// CNC/4 MHT-Function/HLI3_FastMFunctionHandler
FUNCTION_BLOCK HLI3_FastMFunctionHandler
VAR_INPUT
	bForceOff			: BOOL;													(* Forces all bytes in the output array to be 00 and therefore to switch off the digital output *) 
	bReset				: BOOL;													(* Resets the digital output *)
	nFunctionNoOn		: UINT;													(* Specifies the M function number for switching the digital output on *) 
	nDelayOn			: DINT;													(* Specifies a delay time in [µs] for switching on the digital output *)
	nFunctionNoOff		: UINT;													(* Specifies the M function number for switching the digital output off *)
	nDelayOff			: DINT;													(* Specifies a delay time in [µs] for switching off the digital output *)
	stData				: ST_FastMFunctionData;									(* Structure provided by an instance of HLI3_FastMFunctionProvider *)
END_VAR
VAR_OUTPUT
	abyOutput			: ARRAY[0..MAX_FAST_M_FUNC_OUTPUT_IDX] OF BYTE;		(* Output array for a digital oversampling output terminal EL2262 *)  
END_VAR
VAR
	bSwitchOn			: BOOL;
	nSwitchOnOffset		: DINT;
	bSwitchOff			: BOOL;
	nSwitchOffOffset	: DINT;
	bStateChanged		: BOOL;
	bFirstCycle			: BOOL := TRUE;
	byStaticValue		: BYTE;
	byBitmask			: BYTE;
	nBits				: DINT;
	nBytes				: DINT;
	nLoop				: UINT;
	nQueuedCount		: UINT;
	
	eLastState			: E_FastMFunctionState := E_FastMFunctionState.OFF;
	stDequeued			: ST_FastMFunctionBufferItem;
	astQueue			: ARRAY[0..MAX_FAST_M_FUNC_QUEUE_IDX] OF ST_FastMFunctionBufferItem;
	
	fbRtrigReset		: Tc2_Standard.R_TRIG;
	CYCLE_TIME			: UINT := 1000;
END_VAR

(****************************************************************************************)
(* POU:		HLI3_FastMFunctionHandler                     								*)
(* Type:	FB																			*)
(* Author: 	RCH		                                             						*)
(* Date: 	14/10/29																	*)
(* Rev.: 	1.0                                               							*)
(* ------------------------------------------------------------------------------------ *)
(* Desc.:	Function block for handling the oversampled output on an EL2262. The 		*)
(*			output state will be derived from the occurance of two CNC M functions, 	*)
(*			which have to be configured with output method MOS_TS and which have to be	*)
(*			preprocessed by an instance of the HLI3_FastMFunctionProvider function 		*)
(*			block. The switch ON/OFF times can be delayed seperately.					*)					
(*																						*)
(*			THIS FB HAS TO BE CALLED CYCLICALLY IN A 1MS TASK AND THE EL2262 HAS TO 	*)
(*			FEATURE AN OVERSAMPLING FACTOR OF 1000 (125 BYTE) ==> 1µs == 1 bit!!!		*)
(* ------------------------------------------------------------------------------------ *)
(* Rev.:	1.1																			*)
(* Date:	15/05/05								                                   	*)
(* Author:	RCH																		 	*)
(* Desc.:	Fixed issues occured if more than 1 MOS_TS M function was programmed in a   *)
(*			single G-Code block.														*)
(* ------------------------------------------------------------------------------------ *)
(* Rev.:	<Enter revision number here>												*)
(* Date:	<Enter revision data here>				                                   	*)
(* Author:	<Enter author´s shortcut here>											 	*)
(* Desc.:	<Enter description here>													*)
(****************************************************************************************)

(****************************************************************************************)
(*	  						  Refresh buffered switch times 							*)
(****************************************************************************************)
THIS^.RefreshQueue(CYCLE_TIME);

(****************************************************************************************)
(*	  							 	  Reset output										*)
(****************************************************************************************)
fbRtrigReset(CLK:= bReset);

IF fbRtrigReset.Q THEN
	THIS^.ClearQueue();
	bStateChanged				:= TRUE;
	eLastState					:= E_FastMFunctionState.OFF;
END_IF

(****************************************************************************************)
(*	  					    Search for new switch on/off events 						*)
(****************************************************************************************)
bSwitchOn						:= FALSE;
nSwitchOnOffset					:= 0;
bSwitchOff						:= FALSE;
nSwitchOffOffset				:= 0;
nLoop							:= 0;

IF (stData.nFunctionCount > 0) AND (stData.bDataValid) THEN
	REPEAT
		IF (stData.astItem[nLoop].nFunctionNo = nFunctionNoOn) THEN
			bSwitchOn			:= TRUE;
			nSwitchOnOffset		:= stData.astItem[nLoop].nOffset;
		ELSIF (stData.astItem[nLoop].nFunctionNo = nFunctionNoOff) THEN
			bSwitchOff			:= TRUE;
			nSwitchOffOffset	:= stData.astItem[nLoop].nOffset;
		END_IF
	
		nLoop					:= nLoop + 1;
		
		UNTIL ((bSwitchOn AND bSwitchOff) OR (nLoop >= stData.nFunctionCount))
	END_REPEAT	
END_IF

(****************************************************************************************)
(*	  		Buffer found switch on/off events with correspondent switch times			*)
(****************************************************************************************)
IF bSwitchOn AND bSwitchOff THEN
	(* In case switch on and off events have been transmitted within the same cycle, 	*)
	(* order them according to their switch times!										*)
	IF ((nSwitchOnOffset + nDelayOn) < (nSwitchOffOffset + nDelayOff)) THEN
		THIS^.Enqueue(E_FastMFunctionState.ON, nSwitchOnOffset + nDelayOn);
		THIS^.Enqueue(E_FastMFunctionState.OFF, nSwitchOffOffset + nDelayOff); 
	ELSE
		THIS^.Enqueue(E_FastMFunctionState.OFF, nSwitchOffOffset + nDelayOff);
		THIS^.Enqueue(E_FastMFunctionState.ON, nSwitchOnOffset + nDelayOn);
	END_IF
ELSIF bSwitchOn THEN
	THIS^.Enqueue(E_FastMFunctionState.ON, nSwitchOnOffset + nDelayOn);
ELSIF bSwitchOff THEN
	THIS^.Enqueue(E_FastMFunctionState.OFF, nSwitchOffOffset + nDelayOff);
END_IF

(****************************************************************************************)
(*	  				  Set output array according to latest switch state					*)
(****************************************************************************************)
IF bStateChanged OR bFirstCycle THEN
	bStateChanged				:= FALSE;

	IF (eLastState = E_FastMFunctionState.OFF) THEN
		byStaticValue			:= 16#00;
	ELSIF (eLastState = E_FastMFunctionState.ON) THEN
		byStaticValue			:= 16#FF;
	END_IF
	
	Tc2_System.MEMSET(ADR(abyOutput[0]), byStaticValue, SIZEOF(abyOutput));
END_IF

(****************************************************************************************)
(*	  					  Dequeue switch events from the buffer							*)
(****************************************************************************************)
WHILE THIS^.DequeuingRequired DO
	stDequeued					:= THIS^.Dequeue();
	nBits 						:= stDequeued.nSwitchTime MOD 8;
	nBytes 						:= stDequeued.nSwitchTime / 8;
	bStateChanged				:= TRUE;
	IF (stDequeued.nSwitchTime < 0) OR (stDequeued.nSwitchTime > 1000) THEN
		;
	ELSE
		IF ((stDequeued.eState = E_FastMFunctionState.ON) AND (eLastState = E_FastMFunctionState.OFF)) THEN
			byBitmask			:= SHL(BYTE#255, nBits);
			abyOutput[nBytes]	:= abyOutput[nBytes] OR byBitmask;
			eLastState			:= E_FastMFunctionState.ON;
			Tc2_System.MEMSET(ADR(abyOutput[nBytes + 1]), 16#FF, MAX_FAST_M_FUNC_OUTPUT_IDX - nBytes);
		ELSIF ((stDequeued.eState = E_FastMFunctionState.OFF) AND (eLastState = E_FastMFunctionState.ON)) THEN
			byBitmask			:= SHR(BYTE#255, 8 - nBits);
			abyOutput[nBytes]	:= abyOutput[nBytes] AND byBitmask;
			eLastState			:= E_FastMFunctionState.OFF;
			Tc2_System.MEMSET(ADR(abyOutput[nBytes + 1]), 16#00, MAX_FAST_M_FUNC_OUTPUT_IDX - nBytes);
		END_IF
	END_IF
END_WHILE

(****************************************************************************************)
(*	  							   Reset first cycle indicator							*)
(****************************************************************************************)
bFirstCycle						:= FALSE;

METHOD ClearQueue
Tc2_System.MEMSET(ADR(astQueue), 16#00, SIZEOF(astQueue));
nQueuedCount := 0;
END_METHOD

METHOD Dequeue : ST_FastMFunctionBufferItem
VAR
	stReturn	: ST_FastMFunctionBufferItem;
END_VAR
IF (nQueuedCount > 0) THEN
	stReturn		:=	astQueue[0]; 
	Tc2_System.MEMMOVE(ADR(astQueue[0]), ADR(astQueue[1]), SIZEOF(astQueue) - SIZEOF(stReturn));
	
	nQueuedCount	:= nQueuedCount - 1;
	Dequeue			:= stReturn;
END_IF
END_METHOD

PROPERTY DequeuingRequired : BOOL
GET
DequeuingRequired	:= (nQueuedCount > 0) AND 
					   (astQueue[0].eState <> E_FastMFunctionState.EMPTY) AND
					   (astQueue[0].nSwitchTime < CYCLE_TIME);
END_GET
END_PROPERTY

METHOD Enqueue
VAR_INPUT
	eState			: E_FastMFunctionState;
	nSwitchTime		: DINT;
END_VAR
IF (nQueuedCount <= MAX_FAST_M_FUNC_OUTPUT_IDX) THEN
	astQueue[nQueuedCount].eState		:= eState;
	astQueue[nQueuedCount].nSwitchTime	:= nSwitchTime;
	nQueuedCount						:= nQueuedCount + 1;
END_IF
END_METHOD

METHOD RefreshQueue
VAR_INPUT
	nCycleTime: UINT;
END_VAR
IF (nQueuedCount > 0) THEN
	FOR nLoop := 0 TO (nQueuedCount - 1) DO
		astQueue[nLoop].nSwitchTime	:= astQueue[nLoop].nSwitchTime - nCycleTime;
	END_FOR
END_IF
END_METHOD

END_FUNCTION_BLOCK

// CNC/4 MHT-Function/HLI3_FastMFunctionProvider
FUNCTION_BLOCK HLI3_FastMFunctionProvider
VAR_INPUT
	nHliChanIdx				: UINT;													(* HLI channel index of the channel to check for new M functions *)
	anMFunctionNo			: ARRAY[0..MAX_FAST_M_FUNC_ITEM_IDX] OF UINT;			(* List of M functions munbers to handle *)
END_VAR
VAR_OUTPUT
	stData					: ST_FastMFunctionData;									(* Output structure containing informatione about the handled M functions and their execution offsets *)
	bUnknownChannelIndex	: BOOL;													(* TRUE if the given nHliChanIdx is unknown *)
END_VAR
VAR
	bExitAll				: BOOL;
	bFirstCycle				: BOOL := TRUE;
	byTaskIndex				: BYTE;
	nConfiguredFunctions	: UINT;
	nFunctionCount			: UINT;
	nLoop1					: UINT;
	nLoop2					: UINT;
	anMFunctionNoOld		: ARRAY[0..MAX_FAST_M_FUNC_ITEM_IDX] OF UINT;
	pChan					: POINTER TO HIGH_LEVEL_INTERFACE_CH;
	pData					: POINTER TO ST_FastMFunctionItem;
	pTechno					: POINTER TO Techno_Unit_Ch;
	pMHTechno				: POINTER TO HLI_M_H_Prozess;
	
	fbGetTaskIndex			: Tc2_System.GETCURTASKINDEX;
END_VAR

(****************************************************************************************)
(* POU:		HLI3_FastMFunctionProvider                     								*)
(* Type:	FB																			*)
(* Author: 	RCH		                                             						*)
(* Date: 	14/10/29																	*)
(* Rev.: 	1.0                                               							*)
(* ------------------------------------------------------------------------------------ *)
(* Desc.:	FB for handling CNC M functions contained in the input array				*)
(*			'anMFunctionNo'. These M functions have to be configured as MOS_TS. Their	*)
(*			metadata will be copied into the output structure 'stData' to be processed	*)
(*			by instances of the FB HLI3_FastMFunctionHandler!							*)				
(*																						*)
(*			THIS FB HAS TO BE CALLED CYCLICALLY IN A 1MS TASK!!!						*)
(* ------------------------------------------------------------------------------------ *)
(* Rev.:	1.1																			*)
(* Date:	15/05/05								                                   	*)
(* Author:	RCH																		 	*)
(* Desc.:	Fixed issues occured if more than 1 MOS_TS M function was programmed in a   *)
(*			single G-Code block.														*)
(* ------------------------------------------------------------------------------------ *)
(* Rev.:	<Enter revision number here>												*)
(* Date:	<Enter revision data here>				                                   	*)
(* Author:	<Enter author´s shortcut here>											 	*)
(* Desc.:	<Enter description here>													*)
(****************************************************************************************)

(****************************************************************************************)
(*	  Read current (PLC) task id and check whether the cycle time has been exceeded		*)
(****************************************************************************************)
IF bFirstCycle THEN
	fbGetTaskIndex
		(index				=> byTaskIndex);
END_IF

(****************************************************************************************)
(*								Initialize output structure								*)
(****************************************************************************************)
Tc2_System.MEMSET(ADR(stData), 16#00, SIZEOF(stData));

stData.bCycleTimeExceeded	:= TwinCAT_SystemInfoVarList._TaskInfo[byTaskIndex].CycleTimeExceeded;
stData.bDataValid			:= FALSE;
stData.nFunctionCount		:= 0;	

(****************************************************************************************)
(*	  					  Check existence of the given channel index					*)
(****************************************************************************************)
IF NOT HLI3_CheckChannelValid(nChannel := nHliChanIdx) THEN
	bUnknownChannelIndex	:=	TRUE; 
	RETURN;
ELSE
	bUnknownChannelIndex	:=	FALSE;
END_IF

(****************************************************************************************)
(*	  				  Determine the number of configured M functions					*)
(****************************************************************************************)
IF (Tc2_System.MEMCMP(ADR(anMFunctionNo), ADR(anMFunctionNoOld), SIZEOF(anMFunctionNo)) <> 0) THEN
	anMFunctionNoOld				:= anMFunctionNo;
	nConfiguredFunctions			:= 0;
	
	FOR nLoop1 := 0 TO MAX_FAST_M_FUNC_ITEM_IDX DO
		IF (anMFunctionNoOld[nLoop1] > 0) THEN
			nConfiguredFunctions	:= nConfiguredFunctions + 1;
		END_IF
	END_FOR
END_IF

(****************************************************************************************)
(*	  					  	Check occurances of M functions								*)
(****************************************************************************************)
stData.bDataValid					:= TRUE;
bFirstCycle							:= FALSE;

IF (gpCh[nHliChanIdx]^.used_units_std_sync_r = 0) THEN
	RETURN;
END_IF

pChan								:= gpCh[nHliChanIdx];
nFunctionCount						:= 0;
nLoop1 								:= 0;

FOR nLoop1 := 0 TO INT_TO_UINT(HLI_TU_CH_STD_SYNC_MAXIDX) DO
	IF pChan^.techno_unit_std_sync[nLoop1].please_rw AND (pChan^.techno_unit_std_sync[nLoop1].fkt_ctrl_r = Tc2_CncHli.HLI_INTF_M_FKT) THEN
		pTechno						:= ADR(pChan^.techno_unit_std_sync[nLoop1]);
		pMHTechno					:= ADR(pTechno^.attribut_r);	
		
		(* Check whether this FB has to handle the current M function *)
		FOR nLoop2 := 0 TO (nConfiguredFunctions - 1) DO
			IF (pMHTechno^.nr = anMFunctionNo[nLoop2]) THEN
				pData				:= ADR(stData.astItem[nFunctionCount]);
				pData^.nFunctionNo	:= anMFunctionNo[nLoop2];
				pData^.nOffset		:= pMHTechno^.zeit;
				pData^.nCycleCount	:= TwinCAT_SystemInfoVarList._TaskInfo[byTaskIndex].CycleCount;
				
				nFunctionCount		:= nFunctionCount + 1;
				
				pTechno^.please_rw	:= FALSE;
				pTechno^.done_w		:= TRUE;		
				EXIT;	
			END_IF					
		END_FOR
		
		IF (nFunctionCount >= nConfiguredFunctions) THEN
			EXIT;
		END_IF
	ELSIF NOT pChan^.techno_unit_std_sync[nLoop1].please_rw THEN
		EXIT;
	END_IF	
END_FOR

stData.nFunctionCount				:= nFunctionCount;

END_FUNCTION_BLOCK

// CNC/4 MHT-Function/HLI3_QuitAxisMFunction
FUNCTION HLI3_QuitAxisMFunction : BOOL
VAR_INPUT
	/// Number of axis 
	nHliAxisIdx: INT;
END_VAR
VAR
	/// Data of a M/H techno unit 
	pMHProcess: POINTER TO HLI_M_H_PROZESS;
	/// Data of a spindle unit 
	pSProcess: POINTER TO HLI_S_PROZESS;
	/// Data of a techno unit 
	pTProcess: POINTER TO HLI_T_PROZESS;
	/// local pointer to Data of actual Axis 
	pAxisData: POINTER TO HIGH_LEVEL_INTERFACE_AX;
	/// local pointer to actual techno unit 
	pActTechnoUnit: POINTER TO TECHNO_UNIT_AX;
	/// loop variable 
	idx: UINT;
	/// Index of axis specific technology function at HLI 
	nTechFctMaxIdx: UINT;
	/// basis id of a tool 
	nToolBasicId: UDINT;
	/// spindle movement command 
	SpdlMoveCmd: UINT;
	/// SpindleRevolution 
	Revolution: UDINT;
	/// SpindleRevolution 
	pRevolution: POINTER TO UDINT;
	/// Number of M-function 
	FuncNr: UDINT;
END_VAR

(* ========================================================= *)
(*    FUN: HLI_QuitAxisMFunction                             *)
(* --------------------------------------------------------- *)
(*   Desc:                                                   *)
(* Author: MK                                                *)
(*   Rev.: 1.1                                               *)
(*   Date: 18.07.2002                                        *)
(*       : 08.04.2005                                        *)
(* ========================================================= *)

HLI3_QuitAxisMFunction := FALSE;
IF NOT (HLI3_CheckAxisValid(nHliAxisIdx := nHliAxisIdx)) THEN
	RETURN;
END_IF


(* get pointer to Axis data *)
pAxisData := gpAx[nHliAxisIdx];

(* test if there are open synchronisations  *)
IF pAxisData^.used_units_std_sync_r > 0 THEN

	nTechFctMaxIdx := pAxisData^.used_units_std_sync_r - 1;

	FOR idx := 0 TO nTechFctMaxIdx DO
	
		(* get pointer to actual techno unit *)
		pActTechnoUnit := ADR(pAxisData^.techno_unit_std_sync[idx]);
	
		(* test if this M-function has to be acknowledged *)
		IF pActTechnoUnit^.please_rw = TRUE AND				(* request from CNC *)
			pActTechnoUnit^.done_w = FALSE					(* not acknowledged *)
		THEN
	
			IF pActTechnoUnit^.fkt_ctrl_r = HLI_INTF_M_FKT THEN
				(* Example: read number of M-function *)
				pMHProcess := ADR(pActTechnoUnit^.attribut_r.data[0]);
				FuncNr := pMHProcess^.nr;
				//ADSLOG(strMsg:='Axis acknowledge of M-function: %d', nDINT:=UDINT_TO_DINT(FuncNr), strArg:='');
			ELSE
				IF pActTechnoUnit^.fkt_ctrl_r = HLI_INTF_SPINDEL THEN (* spindle-fuction *)
					pSProcess := ADR(pActTechnoUnit^.attribut_r.data[0]);
	
					(* Example: read revolution of S-function *)
					Revolution := DINT_TO_UINT(pSProcess^.rev);
					//ADSLOG(strMsg:='Spindle S-function: %d', nDINT:=UDINT_TO_DINT(Revolution), strArg:='');
	
					(* Example: read number of S-function *)
					SpdlMoveCmd := pSProcess^.move_cmd;
					//ADSLOG(strMsg:='Spindle acknowledge of M-function: %d', nDINT:=SpdlMoveCmd, strArg:='');
				ELSE
					ADSLOGDINT( msgCtrlMask :=    ADSLOG_MSGTYPE_MSGBOX
					                           OR ADSLOG_MSGTYPE_LOG,
								msgFmtStr   := 'Axis acknowledge unknown type: %d',
								dintArg     := pActTechnoUnit^.fkt_ctrl_r);
				END_IF
			END_IF
	
			(* acknowledge this M-function *)
			pActTechnoUnit^.please_rw := FALSE;
			pActTechnoUnit^.done_w := TRUE;
	
			HLI3_QuitAxisMFunction := TRUE;
		END_IF
	END_FOR

END_IF

END_FUNCTION

// CNC/5 Variables/FB_ReadCNCVariables
FUNCTION_BLOCK FB_ReadCNCVariables
VAR_INPUT
	bEnable		:	BOOL ;	(* B *)
	nChanIdx	:   INT;
	eVariablesType : E_CNCVariablesType;
	tIntervall	:   TIME;
END_VAR

VAR_OUTPUT
	Done			:	BOOL;	(* B *)
	Busy			: 	BOOL;	(* E *)	
	Error			:	BOOL;	(* B *)
	ErrorID			:	UDINT;	(* E *) 
END_VAR

VAR_IN_OUT
	 stCNCVariablesViewer_Data : ARRAY[0..MAX_CNC_VAR_LIST_IDX] OF ST_CNCVariablesViewer_Data;
END_VAR

VAR	
	fbTrigger :	R_TRIG;
	fbReadNumber: ADSREAD;
	nParameterNumber : DINT;
		
	fbReadWrite: ADSRDWRT;	
	strVarName : STRING(96);	
	fVarValue  : LREAL;    
 	nIndex     : UDINT;
	nListIndex : UDINT;	
	
	nState	: INT;
	fbTimer : TON;

	nReadLength 	   : UDINT;
	
 	IDXOffsNumber	   : UDINT;
	IDXOffsNamebyIndex : UDINT;
	IDXOffsValuebyIndex : UDINT;	
	stCNCVariablesViewer_Data_Temp : ARRAY[0..MAX_CNC_VAR_LIST_IDX] OF ST_CNCVariablesViewer_Data;
		
	nVEType 				: DINT;
	nVESize 	 			: UDINT;
    nVEMaxIndex1 		   	: UDINT; 
    nVEMaxIndex2 		   	: UDINT;
	strVEVarName 			: STRING(255);	
	strVEDisplayVarName		: STRING(255);
	arrVEDescriptionInput  	: ARRAY[0..259] OF BYTE;
	arrVEOutput 			: ARRAY[0..2047] OF BYTE;
			
	nVEArrayIndex       	: UDINT;
	nListIndexArrayStart	: UDINT; 	
	
	strValue            : STRING(799);
			
	dummyBoolean		: BOOL;
	dummySInt			: SINT;
	dummyUSInt			: USINT;
	dummyInt            : INT;
	dummyUInt			: UINT;
	dummyDInt           : DINT;
	dummyUDInt          : UDINT;
	dummyLReal          : LREAL;
	dummyString         : STRING;
	dummyLargeString    : STRING(799);  

	eVariablesTypeOld : E_CNCVariablesType;
	
END_VAR

VAR CONSTANT
	IDXOffsPNumber  : UDINT := 16#2;	
	IDXOffsVLNumber : UDINT := 16#3;
	IDXOffsVPNumber : UDINT := 16#4;
	IDXOffsVSNumber : UDINT := 16#5;
			
	IDXOffsPNamebyIndex : UDINT := 16#1B;
	IDXOffsVLNamebyIndex : UDINT := 16#1E;
	IDXOffsVPNamebyIndex : UDINT := 16#21;
	IDXOffsVSNamebyIndex : UDINT := 16#24;		
	
	IDXOffsPValuebyIndex : UDINT := 16#1D;
	IDXOffsVLValuebyIndex : UDINT := 16#20;
	IDXOffsVPValuebyIndex : UDINT := 16#23;
	IDXOffsVSValuebyIndex : UDINT := 16#26;
	IDXOffsVEValuebyName : UDINT := 16#2E;		
END_VAR

(****************************************************************************************)
(* POU:		ReadCNCVariables                     										*)
(* Type:	FB																			*)
(* Author: 	TV , MiB                                       								*)
(* Date: 	20.01.2016, 19.12.2016														*)
(* Rev.: 	1.0                                              							*)
(* Rev.: 	1.1 MiB VStrings support (up to 800byte)           							*)
(* ------------------------------------------------------------------------------------ *)
(* Desc:	Description																	*)
(****************************************************************************************)

(****************************************************************************************)
(*	FB reads in P, V.P, V.L., V.S., V.E. Parameter from the CNC Kernel via ADS		    *)
(****************************************************************************************)

IF (NOT HLI3_CheckChannelValid(nChannel := nChanIdx)) THEN	
	RETURN; (* A b b r u c h *)
END_IF

IF 	NOT bEnable OR 
	eVariablesType = E_CNCVariablesType.none  OR
	(gpCh[0]^.channel_mc_control.mode_and_state.state_r.mode = HLI_IMCM_MANUAL_MODE AND eVariablesType <> E_CNCVariablesType.VE) OR
	(gpCh[nChanIdx]^.channel_mc_control.mode_and_state.state_r.state <> HLI_IMCM_PROCESS_ACTIVE AND 
	gpCh[nChanIdx]^.channel_mc_control.mode_and_state.state_r.state <>  HLI_IMCM_PROCESS_HOLD AND eVariablesType <> E_CNCVariablesType.VE) 
		
	THEN
		Tc2_System.MEMSET(ADR(stCNCVariablesViewer_Data),0,SIZEOF(stCNCVariablesViewer_Data));
		fbTrigger(CLK:= FALSE);
		nState := 0;  
	ELSE
		fbTrigger(CLK:= TRUE);	
END_IF

IF fbTrigger.Q OR eVariablesTypeOld <> eVariablesType THEN		
	fbReadNumber(READ:= FALSE);
	fbReadWrite(WRTRD:= FALSE);
	nIndex 		:= 1;	
	nListIndex  := 0;
	nState 		:= 1;
	Error		:= FALSE;	(* B *)
	ErrorID		:= 0;		(* E *) 
END_IF

IF nState <> 0 THEN
	Busy := TRUE;
END_IF

CASE nState OF
	
0:
;  
1: 
	Error		:= FALSE;	(* B *)
	ErrorID		:= 0;	(* E *)

	eVariablesTypeOld :=  eVariablesType;
 
	Tc2_System.MEMSET(ADR(stCNCVariablesViewer_Data_Temp),0,SIZEOF(stCNCVariablesViewer_Data_Temp));
	
   	IF (eVariablesType = E_CNCVariablesType.P) THEN
	      IDXOffsNumber 	 	:= IDXOffsPNumber;
		  IDXOffsNamebyIndex 	:= IDXOffsPNamebyIndex;
		  IDXOffsValuebyIndex 	:= IDXOffsPValuebyIndex;
		  nReadLength			:= 8;			  
	ELSIF (eVariablesType = E_CNCVariablesType.VL) THEN
		 IDXOffsNumber 		 	:=  IDXOffsVLNumber;
		 IDXOffsNamebyIndex  	:= IDXOffsVLNameByIndex;
		 IDXOffsValuebyIndex 	:= IDXOffsVLValuebyIndex;
		 nReadLength			:= 8;
	ELSIF (eVariablesType = E_CNCVariablesType.VP) THEN
		 IDXOffsNumber 		 	:=  IDXOffsVPNumber;
		 IDXOffsNamebyIndex  	:= IDXOffsVPNameByIndex;
		 IDXOffsValuebyIndex 	:= IDXOffsVPValuebyIndex;
		 nReadLength			:= 8;
	ELSIF (eVariablesType = E_CNCVariablesType.VS) THEN
		 IDXOffsNumber 		 	:=  IDXOffsVSNumber;
		 IDXOffsNamebyIndex  	:= IDXOffsVSNameByIndex;
		 IDXOffsValuebyIndex 	:= IDXOffsVSValuebyIndex;
		 nReadLength			:= 8;	
   	END_IF
				
	
	IF (eVariablesType <> E_CNCVariablesType.VE) THEN
		fbReadNumber(
			NETID:= , 
			PORT:= 552, 
			IDXGRP:= 16#22300 + INT_TO_UDINT(nChanIdx)+1, 
			IDXOFFS:= IDXOffsNumber, 
			LEN:= 4, 
			DESTADDR:= ADR(nParameterNumber), 
			READ:= TRUE, 
		);
		
		IF NOT fbReadNumber.Busy THEN
			IF fbReadNumber.Err	THEN
				Error := fbReadNumber.ERR;
				ErrorID := fbReadNumber.ERRID;
				nState := 99;
			ELSE			
				nState := nState + 1;				
			END_IF
		END_IF
	ELSE
		nState := 20;
	END_IF

2:	// Read Variablen Name	
	IF nParameterNumber > 0 THEN 
		fbReadWrite(
		NETID:= , 
		PORT:= 552, 
		IDXGRP:= 16#22300 + INT_TO_UDINT(nChanIdx)+1, 
		IDXOFFS:= IDXOffsNamebyIndex, 
		WRITELEN:= 4, 
		READLEN:= 96, 
		SRCADDR:= ADR(nIndex), 
		DESTADDR:=ADR(strVarName), 
		WRTRD:= TRUE);
	
		IF NOT fbReadWrite.Busy THEN
			IF fbReadWrite.Err	THEN
				Error := fbReadWrite.ERR;
				ErrorID := fbReadWrite.ERRID;
				nState := 99;
			ELSE					
				fbReadWrite(WRTRD:= FALSE);	
				nState := 3;							
			END_IF
		END_IF
	
	ELSE	
		nState := 99;
	END_IF
	
	
3:	// Read Variablen Value	P V.L. V.P. V.S	
		fbReadWrite(
		NETID:= , 
		PORT:= 552, 
		IDXGRP:= 16#22300 + INT_TO_UDINT(nChanIdx)+1, 
		IDXOFFS:= IDXOffsValuebyIndex, 
		WRITELEN:= 4, 
		READLEN:= nReadLength, 
		SRCADDR:= ADR(nIndex), 
		DESTADDR:=ADR(fVarValue), 
		WRTRD:= TRUE);
	
		IF NOT fbReadWrite.Busy THEN
			IF fbReadWrite.Err	THEN
				Error := fbReadWrite.ERR;
				ErrorID := fbReadWrite.ERRID;
				nState := 99;
			ELSE
				stCNCVariablesViewer_Data_Temp[nListIndex].strName := strVarName;
				stCNCVariablesViewer_Data_Temp[nListIndex].strValue := LREAL_TO_STRING(fVarValue);		
				nListIndex := nListIndex+1;								
				nState := 4;
			END_IF
		END_IF		
		
		
4:  
	IF nIndex < DINT_TO_UDINT(nParameterNumber) AND (nListIndex <= MAX_CNC_VAR_LIST_IDX) THEN
		fbReadWrite(WRTRD:= FALSE);
		//nListIndex := nListIndex+1; 
		nIndex := nIndex + 1;
		nState := 2;
	ELSE
			fbTimer(IN:=FALSE);
			nState := 60;
	END_IF

20:    	// Read V.E. Variable element number
		arrVEDescriptionInput[0] := 86; // V
		arrVEDescriptionInput[1] := 46; //.
		arrVEDescriptionInput[2] := 69; //E
		
		fbReadWrite(
			NETID:= , 
			PORT:= 552, 
			IDXGRP:= 16#22300 + INT_TO_UDINT(nChanIdx)+1, 
			IDXOFFS:= 16#44, 
			WRITELEN:= 256, 
			READLEN:= 4, 
			SRCADDR:= ADR(arrVEDescriptionInput), 
			DESTADDR:=ADR(nParameterNumber), 
			WRTRD:= TRUE);

			IF NOT fbReadWrite.Busy THEN
				IF fbReadWrite.Err	THEN
					Error := fbReadWrite.ERR;
					ErrorID := fbReadWrite.ERRID;
					nState := 99;
				ELSE
					fbReadWrite(WRTRD:= FALSE);
					IF nParameterNumber > 0 THEN	
						nIndex := 0;		
						nListIndexArrayStart := 0;
						nVEArrayIndex := 0;			
						nState := 21;					
					ELSE			
						fbTimer(IN:=FALSE);
						nState := 60;			
					END_IF
				END_IF	
			END_IF			
			
21:		// Read V.E. Variable description by index
		MEMCPY(ADR(arrVEDescriptionInput),ADR(nIndex),SIZEOF(nIndex));
		arrVEDescriptionInput[4] := 86; // V
		arrVEDescriptionInput[5] := 46; //.
		arrVEDescriptionInput[6] := 69; //E
		
		fbReadWrite(
			NETID:= , 
			PORT:= 552, 
			IDXGRP:= 16#22300 + INT_TO_UDINT(nChanIdx)+1, 
			IDXOFFS:= 16#45, 
			WRITELEN:= 260, 
			READLEN:= 2048, 
			SRCADDR:= ADR(arrVEDescriptionInput), 
			DESTADDR:=ADR(arrVEOutput), 
			WRTRD:= TRUE);
	
		IF NOT fbReadWrite.Busy THEN
			IF fbReadWrite.Err	THEN
				Error := fbReadWrite.ERR;
				ErrorID := fbReadWrite.ERRID;
				nState := 99;
			ELSE
				fbReadWrite(WRTRD:= FALSE);
				
				//MEMCPY(ADR(nHandle),ADR(arrByte3),SIZEOF(nHandle));
				MEMCPY(ADR(nVEType),ADR(arrVEOutput)+4,SIZEOF(nVEType));
				// MEMCPY(ADR(nAccess),ADR(arrByte3)+4+4,SIZEOF(nAccess));
				MEMCPY(ADR(nVESize),ADR(arrVEOutput)+4+4+4,SIZEOF(nVESize));
				MEMCPY(ADR(nVEMaxIndex1),ADR(arrVEOutput)+4+4+4+4,SIZEOF(nVEMaxIndex1));
				IF nVEMaxIndex1 <> 0 THEN
					MEMCPY(ADR(nVEMaxIndex2),ADR(arrVEOutput)+4+4+4+4+4,SIZEOF(nVEMaxIndex2));
					MEMCPY(ADR(strVEVarName),ADR(arrVEOutput)+4+4+4+4+4+4,SIZEOF(strVEVarName));
				ELSE
					MEMCPY(ADR(strVEVarName),ADR(arrVEOutput)+4+4+4+4+4,SIZEOF(strVEVarName));
				END_IF
												
				IF nVEMaxIndex1 > 0 THEN
					nListIndexArrayStart := nListIndex;
					FOR nVEArrayIndex := 0 TO nVEMaxIndex2-1 DO						
						strVEDisplayVarName := CONCAT(strVEVarName,'[');
						strVEDisplayVarName := CONCAT(strVEDisplayVarName,UDINT_TO_STRING(nVEArrayIndex));
						strVEDisplayVarName := CONCAT(strVEDisplayVarName,']');			
						stCNCVariablesViewer_Data_Temp[nListIndex].strName := strVEDisplayVarName;
						IF (nListIndex < MAX_CNC_VAR_LIST_IDX) THEN
							nListIndex := nListIndex+1;
						ELSE
							EXIT;
						END_IF
							
					END_FOR	
					   nVEArrayIndex := 0;
					   nListIndex := nListIndexArrayStart;
					   nState := 25;											
				ELSE			
					nVEArrayIndex := 0;
					stCNCVariablesViewer_Data_Temp[nListIndex].strName := strVEVarName;						
					nState := 25;
				END_IF						
			END_IF
		END_IF	
		
25:		// Read Value By Name	
		IF nVEMaxIndex1 = 0 THEN			
			strVEVarName := stCNCVariablesViewer_Data_Temp[nListIndex].strName;
		ELSE
			strVEVarName := stCNCVariablesViewer_Data_Temp[nListIndex+nVEArrayIndex].strName ;
		END_IF		
							
		fbReadWrite(
		NETID:= , 
		PORT:= 552, 
		IDXGRP:= 16#22300 + INT_TO_UDINT(nChanIdx)+1, 
		IDXOFFS:= 16#48, 
		WRITELEN:= SIZEOF(strVEVarName), 
		READLEN:= 2048, 
		SRCADDR:= ADR(strVEVarName), 
		DESTADDR:=ADR(arrVEOutput), 
		WRTRD:= TRUE);
		
		IF NOT fbReadWrite.Busy THEN
			IF fbReadWrite.Err	THEN
				Error := fbReadWrite.ERR;
				ErrorID := fbReadWrite.ERRID;
				nState := 99;
			ELSE	
						
				IF nVEType = E_VEVariablesType.BOOLEAN THEN 
					MEMCPY(ADR(dummyBoolean),ADR(arrVEOutput),1);
					strValue := BOOL_TO_STRING(dummyBoolean);
				ELSIF nVEType = E_VEVariablesType.UNS08 THEN
					MEMCPY(ADR(dummyUSInt),ADR(arrVEOutput),1);
					strValue := USINT_TO_STRING(dummyUSInt);
				ELSIF nVEType = E_VEVariablesType.SGN08 THEN
					MEMCPY(ADR(dummySInt),ADR(arrVEOutput),1);
					strValue := SINT_TO_STRING(dummySInt);
				ELSIF nVEType = E_VEVariablesType.UNS16 THEN
					MEMCPY(ADR(dummyUInt),ADR(arrVEOutput),2);
					strValue := UINT_TO_STRING(dummyUInt);
				ELSIF nVEType = E_VEVariablesType.SGN16 THEN
					MEMCPY(ADR(dummyInt),ADR(arrVEOutput),2);
					strValue := INT_TO_STRING(dummyInt);
				ELSIF nVEType = E_VEVariablesType.UNS32 THEN
					MEMCPY(ADR(dummyUDInt),ADR(arrVEOutput),4);
					strValue := UDINT_TO_STRING(dummyUDInt);
				ELSIF nVEType = E_VEVariablesType.SGN32 THEN
					MEMCPY(ADR(dummyDInt),ADR(arrVEOutput),4);
					strValue := DINT_TO_STRING(dummyDInt);
				ELSIF nVEType = E_VEVariablesType.REAL64 THEN
					MEMCPY(ADR(dummyLReal),ADR(arrVEOutput),8);
					strValue := LREAL_TO_STRING(dummyLReal);						
				ELSIF nVEType = E_VEVariablesType.VESTRING THEN					 									
					MEMCPY(ADR(dummyLargeString),ADR(arrVEOutput),nVESize-1);
					strValue := dummyLargeString;
				ELSE
					nState := 99;
				END_IF				
				
				nState := 26;	
			END_IF
		END_IF	
		
26:
		stCNCVariablesViewer_Data_Temp[nListIndex+nVEArrayIndex].strValue := strValue;									
										
		IF nVEArrayIndex < nVEMaxIndex2-1 AND  nVEMaxIndex1 <> 0 THEN
			fbReadWrite(WRTRD:= FALSE);
			nVEArrayIndex := nVEArrayIndex +1;
			IF (nListIndex+nVEArrayIndex <= MAX_CNC_VAR_LIST_IDX) THEN
				nState := 25;
			ELSE
				nState := 60;
			END_IF
		ELSE
			IF (nListIndex <= MAX_CNC_VAR_LIST_IDX) THEN
				nListIndex := nListIndex+nVEArrayIndex +1;
				nState := 30;
			ELSE
				nState := 60;
			END_IF		
			
		END_IF
		
30:  
	IF nIndex < DINT_TO_UDINT(nParameterNumber-1) THEN
		fbReadWrite(WRTRD:= FALSE);		 
		nIndex := nIndex + 1;
		nState := 21;
	ELSE
		fbReadWrite(WRTRD:= FALSE);				
		fbTimer(IN:=FALSE);			
		nState := 60;
	END_IF

60:
	// Output
	Tc2_System.MEMCPY(ADR(stCNCVariablesViewer_Data),ADR(stCNCVariablesViewer_Data_Temp),SIZEOF(stCNCVariablesViewer_Data_Temp));
	fbTimer(IN:=TRUE , PT:=tIntervall);	
	IF fbTimer.Q THEN
		fbReadNumber(READ:= FALSE);
		fbReadWrite(WRTRD:= FALSE);
		nListIndex := 0;
		nIndex := 1;
		nState := 1;
	END_IF

99: // Error 
	nIndex := 1;
	nListIndex := 0;
	fbReadNumber(READ:= FALSE);
	fbReadWrite(WRTRD:= FALSE);
	fbTimer(IN:=FALSE);
	nState := 60;			
END_CASE

END_FUNCTION_BLOCK

// CNC/5 Variables/HLI3_GetVEChannelBooleanValue
FUNCTION HLI3_GetVEChannelBooleanValue : BOOL
VAR_INPUT
	/// HLI Channel Index
	nChanIdx: INT;
	/// Index of variable  range 1 ...     HLI_VE_VALUEMAX 
	nVEIndex: DINT;
	/// Array index. 0 if no array 
	nArrayIndex: DINT := 0;
	/// serves acess to the global variable array 
	bGlobal: BOOL;
END_VAR
VAR
	pVeData: POINTER TO VEData := 0;
	/// Size of the datatype of the returned value 
	iDatatypeSize: DINT;
	ptr: POINTER TO BOOL;
	ChIdx: UDINT;
	SizeField: DINT := 0;
END_VAR

(* ========================================================= *)
(*    FUN: GetVEChannelDINTValue                            *)
(* --------------------------------------------------------- *)
(*   Desc: Reads a V.E.Variable of Boolean                   *)
(* 	 Author: CL  / TV                                        *)
(*   Date: 16.05.2006                                        *)
(*   Last: 05.12.2013                                        *)
(*   Rev.: 1.3                                               *)
(* ========================================================= *)

IF  nVEIndex >= 0 AND
	nArrayIndex >= 0 THEN

	(* test if channel specific or global *)
	IF bGlobal = FALSE  THEN
		IF NOT HLI3_CheckChannelValid(nChannel := nChanIdx) THEN
			RETURN;
		END_IF
				
		pVeData := gpVECh[nChanIdx];
	ELSE
		pVeData := gpVEGlobal;
	END_IF

	IF pVeData <> 0 THEN
		IF pVeData <> 0 THEN
			iDatatypeSize := SIZEOF(ptr^);
                         	ptr := pVeData +  24  * nVEIndex + (iDatatypeSize * nArrayIndex);
                           HLI3_GetVEChannelBooleanValue := ptr^; (* successfully completed return *)
                END_IF
	END_IF
END_IF

END_FUNCTION

// CNC/5 Variables/HLI3_GetVEChannelDIntValue
FUNCTION HLI3_GetVEChannelDIntValue : DINT
VAR_INPUT
	/// HLI Channel Index 
	nChanIdx: INT;
	/// Index of variable  range 1 ...     HLI_VE_VALUEMAX 
	nVEIndex: DINT;
	/// Array index. 0 if no array 
	nArrayIndex: DINT := 0;
	/// serves acess to the global variable array 
	bGlobal: BOOL;
END_VAR
VAR
	pVeData: POINTER TO VEData := 0;
	/// Size of the datatype of the returned value 
	iDatatypeSize: DINT;
	ptr: POINTER TO DINT;
	ChIdx: UDINT;
	SizeField: DINT := 0;
END_VAR

(* ========================================================= *)
(*    FUN: GetVEChannelDINTValue                            *)
(* --------------------------------------------------------- *)
(*   Desc: Reads a V.E.Variable of DINT                    *)
(* 	 Author: CL  / TV                                        *)
(*   Date: 16.05.2006                                        *)
(*   Last: 28.01.2013                                        *)
(*   Rev.: 1.3                                               *)
(* ========================================================= *)

IF  nVEIndex >= 0 AND
	nArrayIndex >= 0 THEN

	(* test if channel specific or global *)
	IF bGlobal = FALSE  THEN
		IF NOT HLI3_CheckChannelValid(nChannel := nChanIdx) THEN
			RETURN;
		END_IF
				
		pVeData := gpVECh[nChanIdx];
	ELSE
		pVeData := gpVEGlobal;
	END_IF

	IF pVeData <> 0 THEN
		IF pVeData <> 0 THEN
			iDatatypeSize := SIZEOF(ptr^);
                         	ptr := pVeData +  24  * nVEIndex + (iDatatypeSize * nArrayIndex);
                           HLI3_GetVEChannelDIntValue := ptr^; (* successfully completed return *)
                END_IF
	END_IF
END_IF

END_FUNCTION

// CNC/5 Variables/HLI3_GetVEChannelLRealValue
FUNCTION HLI3_GetVEChannelLRealValue : LREAL
VAR_INPUT
	/// HLI Channel Index
	nChanIdx: INT;
	/// Index of variable  range 1 ...     HLI_VE_VALUEMAX 
	nVEIndex: DINT;
	/// Array index. 0 if no array 
	nArrayIndex: DINT := 0;
	/// serves acess to the global variable array 
	bGlobal: BOOL;
END_VAR
VAR
	pVeData: POINTER TO VEData := 0;
	/// Size of the datatype of the returned value 
	iDatatypeSize: DINT;
	ptr: POINTER TO LREAL;
	ChIdx: UDINT;
	SizeField: DINT := 0;
END_VAR

(* ========================================================= *)
(*    FUN: GetVEChannelLrealValue                            *)
(* --------------------------------------------------------- *)
(*   Desc: Reads a V.E.Variable of REAL64                    *)
(* 	 Author: CL  / TV                                        *)
(*   Date: 16.05.2006                                        *)
(*   Last: 28.01.2013                                        *)
(*   Rev.: 1.3                                               *)
(* ========================================================= *)

IF  nVEIndex >= 0 AND
	nArrayIndex >= 0 THEN

	(* test if channel specific or global *)
	IF bGlobal = FALSE  THEN
		IF NOT HLI3_CheckChannelValid(nChannel := nChanIdx) THEN
			RETURN;
		END_IF
				
		pVeData := gpVECh[nChanIdx];
	ELSE
		pVeData := gpVEGlobal;
	END_IF

	IF pVeData <> 0 THEN
		IF pVeData <> 0 THEN
			iDatatypeSize := SIZEOF(ptr^);
                         	ptr := pVeData +  24  * nVEIndex + (iDatatypeSize * nArrayIndex);
                           HLI3_GetVEChannelLRealValue := ptr^; (* successfully completed return *)
                END_IF
	END_IF
END_IF

END_FUNCTION

// CNC/5 Variables/HLI3_GetVEChannelStringValue
FUNCTION HLI3_GetVEChannelStringValue : STRING(23)
VAR_INPUT
	/// HLI Channel Index
	nChanIdx: INT;
	/// Index of variable  range 1 ...     HLI_VE_VALUEMAX 
	nVEIndex: DINT;
	/// Array index. 0 if no array 
	nArrayIndex: DINT := 0;
	/// serves acess to the global variable array 
	bGlobal: BOOL;
END_VAR
VAR
	pVeData: POINTER TO VEData := 0;
	/// Size of the datatype of the returned value 
	iDatatypeSize: DINT;
	ptr: POINTER TO STRING(24);
	ChIdx: INT;
END_VAR

(* ========================================================= *)
(*    FUN: GetVEChannelStringValue                           *)
(* --------------------------------------------------------- *)
(*   Desc: Reads a V.E.Variable of STRING                    *)
(* 	 Author: CL / TV                                         *)
(*   Date: 16.05.2006                                        *)
(*   Last: 28.01.013                                        *)
(*   Rev.: 1.1                                               *)
(* ========================================================= *)

(* Config Example
	VAR[0].name                                           StringValue
	VAR[0].index                                           1
	VAR[0].TYPE                                           STRING
	VAR[0].scope                                          GLOBAL
	VAR[0].synchronisation                                TRUE
	VAR[0].access_rights                                  READ_WRITE
	VAR[0].array_size                                     21
	VAR[0].size                                           24
	VAR[0].create_hmi_interface                           0
*)

IF  nVEIndex >= 0 AND
	nArrayIndex >= 0 THEN

	(* test if channel specific or global *)
	IF bGlobal = FALSE  THEN
		IF NOT HLI3_CheckChannelValid(nChannel := nChanIdx) THEN
			RETURN;
		END_IF
		pVeData := gpVECh[nChanIdx];
	ELSE
		pVeData := gpVEGlobal;
	END_IF

	IF pVeData <> 0 THEN
		 IF pVeData <> 0 THEN
			iDatatypeSize := SIZEOF(ptr^);
			iDatatypeSize := 24;
            ptr := pVeData +  24  * nVEIndex + (iDatatypeSize * nArrayIndex);
            HLI3_GetVEChannelStringValue := ptr^; (* successfully completed return *)
         END_IF
	END_IF
END_IF

END_FUNCTION

// CNC/5 Variables/HLI3_LinkVEChannelStructure
FUNCTION HLI3_LinkVEChannelStructure : POINTER TO DWORD
VAR_INPUT
	/// HLI Channel Index 
	nChanIdx: INT;	
	/// serves acess to the global variable array 
	bGlobal: BOOL;
END_VAR
VAR
	pVeData: POINTER TO VEData := 0;
	ptr: POINTER TO DWORD;
	ChIdx: UDINT;
	nVEIndex: POINTER TO DWORD;
END_VAR

(* ========================================================= *)
(*    FUN: LinkVEChannelStructure                            *)
(* --------------------------------------------------------- *)
(*   Desc: Link VE variable to the memory of the CNC         *)
(*   Author: CL, MK                                            *)
(*   Date: 16.05.2006                                        *)
(*   Rev.: 1.3                                               *)
(*       : MK  access changed                                *)
(*		   1.2												 *)
(*		   MiB 7.11.2012 check zero pointers				 *)
(*		   TV 19.08.2015 Input Parm. nIndex removed          *) 
(* ========================================================= *)

	(* test if channel specific or global *)
     IF bGlobal THEN
    	IF gpVEGlobal = 0  THEN   (* check for  zero pointer *)
        	RETURN; (* Cancel *)
        END_IF
			pVeData := gpVEGlobal;
	 ELSE
		IF NOT HLI3_CheckChannelValid(nChannel := nChanIdx) THEN
			RETURN;
		END_IF
							
		pVeData := gpVECh[nChanIdx];
	END_IF 

	IF pVeData <> 0 THEN
    	ptr := pVeData;
		HLI3_LinkVEChannelStructure := ptr; (* successfully completed return *)
	END_IF

END_FUNCTION

// CNC/5 Variables/HLI3_SetVEChannelBooleanValue
FUNCTION HLI3_SetVEChannelBooleanValue : BOOL
VAR_INPUT
	/// HLI Channel Index
	nChanIdx: INT;
	/// Index of variable  range 1 ...     HLI_VE_VALUEMAX 
	nVEIndex: DINT;
	/// Array index. 0 if no array 
	nArrayIndex: DINT := 0;
	/// serves acess to the global variable array 
	bGlobal: BOOL;
	/// Value to be written 
	val: BOOL;
END_VAR
VAR
	pVeData: POINTER TO VEData := 0;
	/// Size of the datatype of the returned value 
	iDatatypeSize: DINT;
	ptr: POINTER TO BOOL;
	ChIdx: UDINT;
	SizeField: DINT := 0;
END_VAR

(* ========================================================= *)
(*    FUN: SetVEChannelDIntValue                           *)
(* --------------------------------------------------------- *)
(*   Desc: Writes a V.E.Variable of REAL64                    *)
(* 	 Author: CL  / TV                                        *)
(*   Date: 16.05.2006                                        *)
(*   Last: 05.12.2013                                        *)
(*   Rev.: 1.3                                               *)
(* ========================================================= *)

IF  nVEIndex >= 0 AND
	nArrayIndex >= 0 THEN

	(* test if channel specific or global *)
	IF bGlobal = FALSE  THEN
		IF NOT HLI3_CheckChannelValid(nChannel := nChanIdx) THEN
			RETURN;
		END_IF
				
		pVeData := gpVECh[nChanIdx];
	ELSE
		pVeData := gpVEGlobal;
	END_IF

	IF pVeData <> 0 THEN
		IF pVeData <> 0 THEN
			iDatatypeSize := SIZEOF(ptr^);
            ptr := pVeData +  24  * nVEIndex + (iDatatypeSize * nArrayIndex);
			ptr^:=val;
            HLI3_SetVEChannelBOOLeanValue := TRUE; (* successfully completed return *)						  						   
       	END_IF
	END_IF
END_IF

END_FUNCTION

// CNC/5 Variables/HLI3_SetVEChannelDIntValue
FUNCTION HLI3_SetVEChannelDIntValue : BOOL
VAR_INPUT
	/// HLI Channel Index
	nChanIdx: INT;
	/// Index of variable  range 1 ...     HLI_VE_VALUEMAX 
	nVEIndex: DINT;
	/// Array index. 0 if no array 
	nArrayIndex: DINT := 0;
	/// serves acess to the global variable array 
	bGlobal: BOOL;
	/// Value to be written 
	val: DINT;
END_VAR
VAR
	pVeData: POINTER TO VEData := 0;
	/// Size of the datatype of the returned value 
	iDatatypeSize: DINT;
	ptr: POINTER TO DINT;
	ChIdx: UDINT;
	SizeField: DINT := 0;
END_VAR

(* ========================================================= *)
(*    FUN: SetVEChannelDIntValue                           *)
(* --------------------------------------------------------- *)
(*   Desc: Writes a V.E.Variable of REAL64                    *)
(* 	 Author: CL  / TV                                        *)
(*   Date: 16.05.2006                                        *)
(*   Last: 28.01.2013                                        *)
(*   Rev.: 1.3                                               *)
(* ========================================================= *)

IF  nVEIndex >= 0 AND
	nArrayIndex >= 0 THEN

	(* test if channel specific or global *)
	IF bGlobal = FALSE  THEN
		IF NOT HLI3_CheckChannelValid(nChannel := nChanIdx) THEN
			RETURN;
		END_IF
				
		pVeData := gpVECh[nChanIdx];
	ELSE
		pVeData := gpVEGlobal;
	END_IF

	IF pVeData <> 0 THEN
		IF pVeData <> 0 THEN
			iDatatypeSize := SIZEOF(ptr^);
            ptr := pVeData +  24  * nVEIndex + (iDatatypeSize * nArrayIndex);
			ptr^:=val;
            HLI3_SetVEChannelDIntValue := TRUE; (* successfully completed return *)						  						   
       	END_IF
	END_IF
END_IF

END_FUNCTION

// CNC/5 Variables/HLI3_SetVEChannelLRealValue
FUNCTION HLI3_SetVEChannelLRealValue : BOOL
VAR_INPUT
	/// HLI Channel Index
	nChanIdx: INT;
	/// Index of variable  range 1 ...     HLI_VE_VALUEMAX 
	nVEIndex: DINT;
	/// Array index. 0 if no array 
	nArrayIndex: DINT := 0;
	/// serves acess to the global variable array 
	bGlobal: BOOL;
	/// Value to be written 
	val: LREAL;
END_VAR
VAR
	pVeData: POINTER TO VEData := 0;
	/// Size of the datatype of the returned value 
	iDatatypeSize: DINT;
	ptr: POINTER TO LREAL;
	ChIdx: UDINT;
	SizeField: DINT := 0;
END_VAR

(* ========================================================= *)
(*    FUN: SetVEChannelLrealValue                           *)
(* --------------------------------------------------------- *)
(*   Desc: Writes a V.E.Variable of REAL64                    *)
(* 	 Author: CL  / TV                                        *)
(*   Date: 16.05.2006                                        *)
(*   Last: 06.03.2012                                        *)
(*   Rev.: 1.3                                               *)
(* ========================================================= *)

IF  nVEIndex >= 0 AND
	nArrayIndex >= 0 THEN

	(* test if channel specific or global *)
	IF bGlobal = FALSE  THEN
		IF NOT HLI3_CheckChannelValid(nChannel := nChanIdx) THEN
			RETURN;
		END_IF
				
		pVeData := gpVECh[nChanIdx];
	ELSE
		pVeData := gpVEGlobal;
	END_IF

	IF pVeData <> 0 THEN
		IF pVeData <> 0 THEN
			iDatatypeSize := SIZEOF(ptr^);
            ptr := pVeData +  24  * nVEIndex + (iDatatypeSize * nArrayIndex);
			ptr^:=val;
            HLI3_SetVEChannelLRealValue := TRUE; (* successfully completed return *)						  						   
       	END_IF
	END_IF
END_IF

END_FUNCTION

// CNC/5 Variables/HLI3_SetVEChannelStringValue
FUNCTION HLI3_SetVEChannelStringValue : BOOL
VAR_INPUT
	/// HLI Channel Index
	nChanIdx: INT;
	/// Index of variable  range 1 ...     HLI_VE_VALUEMAX 
	nVEIndex: DINT;
	/// Array index. 0 if no array 
	nArrayIndex: DINT := 0;
	/// Value to be written 
	val: STRING(23);
	/// serves acess to the global variable array 
	bGlobal: BOOL;
END_VAR
VAR
	pVeData: POINTER TO VEData := 0;
	/// Size of the datatype of the returned value 
	iDatatypeSize: DINT;
	ptr: POINTER TO STRING;
	ChIdx: INT;
END_VAR

(* ========================================================= *)
(*    FUN: SetVEChannelStringValue                           *)
(* --------------------------------------------------------- *)
(*   Desc: Writes a V.E.Variable of STRING                   *)
(* 	 Author: CL / TV                                         *)
(*   Date: 16.05.2006                                        *)
(*   Last : 13.12.2012										 *)
(*   Rev.: 1.1                                               *)
(* ========================================================= *)

(* Config Example
	VAR[0].name                                           StringValue
	VAR[0].index                                           1
	VAR[0].TYPE                                           STRING
	VAR[0].scope                                          GLOBAL
	VAR[0].synchronisation                                TRUE
	VAR[0].access_rights                                  READ_WRITE
	VAR[0].array_size                                     21
	VAR[0].size                                           24
	VAR[0].create_hmi_interface                           0
*)

IF  nVEIndex >= 0 AND
	nArrayIndex >= 0 THEN

	(* test if channel specific or global *)
	IF bGlobal = FALSE  THEN
		IF NOT HLI3_CheckChannelValid(nChannel := nChanIdx) THEN
			RETURN;
		END_IF
				
		pVeData := gpVECh[nChanIdx];
	ELSE
		pVeData := gpVEGlobal;
	END_IF

	IF pVeData <> 0 THEN
		iDatatypeSize := SIZEOF(ptr^);
		iDatatypeSize := 24;
        ptr := ADR(pVeData^)  +  24  * nVEIndex + (iDatatypeSize * (nArrayIndex));
        ptr^ := val; (* successfully completed return *)
		HLI3_SetVEChannelStringValue := TRUE;
	END_IF
END_IF

END_FUNCTION

// CNC/6 BlockSearch/HLI3_BlockSearch
FUNCTION_BLOCK HLI3_BlockSearch
VAR_INPUT
	/// Number of channel 
	nChanIdx: INT;
	/// interface values 
	BlockSearch: ST_BlockSearch;
END_VAR
VAR_IN_OUT
	/// Edge signal 
	bStartWrite: BOOL;
	/// Edge signal 
	bStartRead: BOOL;
END_VAR
VAR_OUTPUT
	Busy: BOOL;
	Err: BOOL;
	nErrorState: UINT;
	/// interface values 
	nActType: INT;
	fActDistance: LREAL;
	bActAutoReturn: BOOL;
	nActDeviationMax: UDINT;
	nActBlockNumber: DINT;
	nActPass: DINT;
	nActBlockCount: DINT;
	/// current values 
	actualBlockNumber: DINT := 0;
	actualBlockCount: UDINT := 0;
	actualBlockCount_AfterReset: UDINT := 0;
	coveredDistance: DINT;
	coveredDistance_AfterReset: DINT := 0;
END_VAR
VAR
	bReadStarted: BOOL;
	bWriteStarted: BOOL;
	rtStartRead: R_TRIG;
	rtStartWrite: R_TRIG;
	writeType: WriteBsType;
	readType: ReadBsType;
	writeDistance: WriteBsCoveredDistance;
	readDistance: ReadBsCoveredDistance;
	writeAutoReturn: WriteBsAutoReturn;
	readAutoReturn: ReadBsAutoReturn;
	writeDeviationMax: WriteBsDeviationMax;
	readDeviationMax: ReadBsDeviationMax;
	writeBlockNumber: WriteBsBlockNumber;
	ReadBlockNumber: ReadBsBlockNumber;
	writeBlockCount: WriteBsBlockCount;
	ReadBlockCount: ReadBsBlockCount;	
	writePass: WriteBsPass;
	readPass: ReadBsPass;
	nChannelIdxGrp: UDINT;
	/// Timer to read axisposition cyclically        
	Timer: TON;
	actualcoveredDistance: BOOL;
	ChannelMode: UDINT;
	BlockSearchStart: BOOL;
END_VAR

(* ---------------------*----------------------------------|------------------------------------------------------- *)
(* PURPOSE:                                                                                                         *)
(*                                                                                                                  *)
(*                                                                                                                  *)
(* SCOPE:                                                                                                           *)
(*                                                                                                                  *)
(*                                                                                                                  *)
(* REMARKS:                                                                                                         *)
(*                                                                                                                  *)
(*                                                                                                                  *)
(* AUTHOR:              VERSION     DATE                   CHECKED FROM      DATE     STATUS                        *)
(*    MK                1.0         07.05.2003                                                                      *)
(*    TV                1.1         10.06.2006                                                                      *)
(*    TV                1.2         20.08.2014                                                                      *)
(*    TV                1.2         29.09.2014                                                                      *)
(*    TV                1.3         25.06.2015                                                                      *)
(* ---------------------*----------------------------------|------------------------------------------------------- *)

IF NOT HLI3_CheckChannelValid(nChannel := nChanIdx) THEN
	RETURN;
END_IF




Err := FALSE;
nChannelIdxGrp := 16#00020100 + INT_TO_UDINT(nChanIdx)+1;
BlockSearchStart := FALSE;


(* ----------------------------------- *)
(* --- write block search commands --- *)
(* ----------------------------------- *)

rtStartWrite(CLK:=bStartWrite);
IF rtStartWrite.Q THEN
   bWriteStarted := TRUE;
   bStartWrite := FALSE; (* reset the HMI signal *)
END_IF

IF bWriteStarted THEN
   Busy := TRUE;
   IF BlockSearch.nType = 5 THEN
   	BlockSearch.nType := 3;								(* start position by block count *)

		BlockSearch.bAutoReturn := TRUE;
		(*nPass	:= 1;*)
	END_IF

	(* write block search data to memory *)
   writeType(nIdxGrp:=nChannelIdxGrp, bStart:=rtStartWrite.Q, nType:=BlockSearch.nType);
   writeDistance(nIdxGrp:=nChannelIdxGrp, bStart:=rtStartWrite.Q, fDistance:=(BlockSearch.fDistance*10.0));
   writeAutoReturn(nIdxGrp:=nChannelIdxGrp, bStart:=rtStartWrite.Q, bAutoReturn:=BlockSearch.bAutoReturn);
   writeDeviationMax(nIdxGrp:=nChannelIdxGrp, bStart:=rtStartWrite.Q, nDeviationMax:=BlockSearch.nDeviationMax);
   writePass(nIdxGrp:=nChannelIdxGrp, bStart:=rtStartWrite.Q, nPass:=BlockSearch.nPass);

	CASE BlockSearch.nType OF		(* count and number share a part of the memory *)
		3: writeBlockCount(nIdxGrp:=nChannelIdxGrp, bStart:=rtStartWrite.Q, nBlockCount:=BlockSearch.nBlockCount);
		4: writeBlockNumber(nIdxGrp:=nChannelIdxGrp, bStart:=rtStartWrite.Q, nBlockNumber:=BlockSearch.nBlockNumber);
   END_CASE

   IF writeType.Busy = FALSE
      AND writeDistance.BUSY = FALSE
      AND writeAutoReturn.BUSY = FALSE
      AND writeDeviationMax.BUSY = FALSE
      AND writeBlockNumber.BUSY = FALSE
      AND writePass.BUSY = FALSE
      AND writeBlockCount.BUSY = FALSE
   THEN
      Busy := FALSE;
      bWriteStarted := FALSE;
      BlockSearchStart := TRUE;
   END_IF
END_IF


(* Satzsuchlauf starten *)

(*
IF (BlockSearchStart) AND ((nType = 3) OR (nType = 4)) THEN
	PLCMachineMode[nChan].Start := TRUE;
END_IF
*)

(* -------------------------------- *)
(* --- read block search states --- *)
(* -------------------------------- *)

(* the next rows only for test *)
(* Start a cyclic timer with period 2 sec. *)
Timer(IN := NOT(Timer.Q), PT := T#2000ms);

rtStartRead(CLK:=bStartRead);
(*rtStartRead(CLK:=Timer.Q);*)
IF rtStartRead.Q THEN
   bReadStarted := TRUE;
END_IF

IF bReadStarted THEN
	Busy := TRUE;

   readType(nIdxGrp:=nChannelIdxGrp, bStart:=rtStartRead.Q, pDest:=ADR(nActType));
   readDistance(nIdxGrp:=nChannelIdxGrp, bStart:=rtStartRead.Q, pDest:=ADR(fActDistance));
   readAutoReturn(nIdxGrp:=nChannelIdxGrp, bStart:=rtStartRead.Q, pDest:=ADR(bActAutoReturn));
   readDeviationMax(nIdxGrp:=nChannelIdxGrp, bStart:=rtStartRead.Q, pDest:=ADR(nActDeviationMax));
	CASE nActType OF			(* count and number cannot be read within a single cycle! *)
		3: readBlockCount(nIdxGrp:=nChannelIdxGrp, bStart:=rtStartRead.Q, pDest:=ADR(nActBlockCount));
		4: readBlockNumber(nIdxGrp:=nChannelIdxGrp, bStart:=rtStartRead.Q, pDest:=ADR(nActBlockNumber));
	END_CASE;
   readPass(nIdxGrp:=nChannelIdxGrp, bStart:=rtStartRead.Q, pDest:=ADR(nActPass));

   (*
   readActualBlockNumber(nIdxGrp:=nChannelIdxGrp, bStart:=rtStartRead.Q, pDest:=ADR(actualBlockNumber));
   readActualBlockCount(nIdxGrp:=nChannelIdxGrp, bStart:=rtStartRead.Q, pDest:=ADR(actualBlockCount));
   *)

   IF readType.Busy = FALSE
      AND readDistance.Busy = FALSE
      AND readAutoReturn.Busy = FALSE
      AND readDeviationMax.Busy = FALSE
      AND readBlockNumber.Busy = FALSE
      AND readPass.Busy = FALSE      
   THEN
		Busy := FALSE;

		bReadStarted := FALSE;
		bStartRead := FALSE; (* reset the HMI signal *)
   END_IF
END_IF

actualBlockNumber := gpCh[nChanIdx]^.bahn_state.block_nr_r;
actualBlockCount  := gpCh[nChanIdx]^.bahn_state.block_count_r; 

coveredDistance := gpCh[nChanIdx]^.bahn_state.covered_distance_r;  (* just read actual covered distance *)

(* Speichert die Unterbrechungsstelle *)
ChannelMode := HLI3_GetChannelMode(nChanIdx);
IF (actualBlockCount <> 0) AND (ChannelMode = 2) AND (CNCSystem.Channel[nChanIdx].ActState =4) THEN
	actualBlockCount_AfterReset := actualBlockCount;									(* Zeiger bleibt auch nach Reset erhalten *)
	coveredDistance_AfterReset := coveredDistance;
END_IF

(*	UnterbrechungsstelleWeg			:= coveredDistance/10.0;*)

(*actualBlockNumber := gpAx[0]^.lr_state.block_nr_r;  asume first axis is always moved *)


(* handshake during block search on/off *)
gpCh[nChanIdx]^.bahn_lc_control.block_search.enable_w := TRUE;

IF gpCh[nChanIdx]^.bahn_lc_control.block_search.command_r <>
   gpCh[nChanIdx]^.bahn_lc_control.block_search.state_w THEN

   (* acknowledge *)
   gpCh[nChanIdx]^.bahn_lc_control.block_search.state_w :=
      gpCh[nChanIdx]^.bahn_lc_control.block_search.command_r;

(*
   (* pup up of change *)
   IF gpCh[nHliChIfcIdx]^.bahn_lc_control.block_search.state_w THEN
      ADSLOGDINT( msgCtrlMask := ADSLOG_MSGTYPE_MSGBOX OR ADSLOG_MSGTYPE_LOG,
                  msgFmtStr := 'block search: %d', dintArg := 1);
   ELSE
      ADSLOGDINT( msgCtrlMask := ADSLOG_MSGTYPE_MSGBOX OR ADSLOG_MSGTYPE_LOG,
                  msgFmtStr := 'block search: %d', dintArg := 0);
   END_IF
*)
END_IF

END_FUNCTION_BLOCK

// CNC/6 BlockSearch/ReadBlockCount
FUNCTION_BLOCK ReadBlockCount
VAR_INPUT
	nIdxGrp: UDINT;
	bStart: BOOL;
	pDest: POINTER TO DINT;
END_VAR
VAR_OUTPUT
	Busy: BOOL;
	bErr: BOOL;
END_VAR
VAR
	fbRead: ADSREAD;
	bStarted: BOOL;
END_VAR

IF bStarted = FALSE THEN
   IF bStart = TRUE THEN
      bStarted := TRUE;
      bErr := FALSE;
      Busy := TRUE;
   END_IF
END_IF

IF bStarted THEN
   (* raising edge of Timer triggers read request *)
   fbRead( NetID := '', Port := 553, IdxGrp := nIdxGrp, IdxOffs := 16#0000000D,
         LEN := 4, DestAddr := pDest, READ := bStarted, TMOUT := T#1s);
   IF NOT fbRead.Busy THEN
      (* There was an error in the execution of the read request *)
      IF fbRead.Err THEN
         bErr := TRUE;
      END_IF
      fbRead(READ := FALSE);    (* reset because of edge detection in FB ADSREAD *)
      bStarted := FALSE;
      Busy := FALSE;
   END_IF
END_IF

END_FUNCTION_BLOCK

// CNC/6 BlockSearch/ReadBlockNumber
FUNCTION_BLOCK ReadBlockNumber
VAR_INPUT
	nIdxGrp: UDINT;
	bStart: BOOL;
	pDest: POINTER TO DINT;
END_VAR
VAR_OUTPUT
	Busy: BOOL;
	bErr: BOOL;
END_VAR
VAR
	fbRead: ADSREAD;
	bStarted: BOOL;
END_VAR

IF bStarted = FALSE THEN
   IF bStart = TRUE THEN
      bStarted := TRUE;
      bErr := FALSE;
      Busy := TRUE;
   END_IF
END_IF

IF bStarted THEN
   (* raising edge of Timer triggers read request *)
   fbRead( NetID := '', Port := 553, IdxGrp := nIdxGrp, IdxOffs := 16#0000000E,
         LEN := 4, DestAddr := pDest, READ := bStarted, TMOUT := T#1s);
   IF NOT fbRead.Busy THEN
      (* There was an error in the execution of the read request *)
      IF fbRead.Err THEN
         bErr := TRUE;
      END_IF
      fbRead(READ := FALSE);    (* reset because of edge detection in FB ADSREAD *)
      bStarted := FALSE;
      Busy := FALSE;
   END_IF
END_IF

END_FUNCTION_BLOCK

// CNC/6 BlockSearch/WriteBsType
FUNCTION_BLOCK WriteBsType
VAR_INPUT
	nIdxGrp: UDINT;
	bStart: BOOL;
	nType: UINT;
END_VAR
VAR_OUTPUT
	Busy: BOOL;
	bErr: BOOL;
END_VAR
VAR
	fbWrite: ADSWRITE;
	bStarted: BOOL;
END_VAR

IF bStarted = FALSE THEN
   IF bStart = TRUE THEN
      bStarted := TRUE;
      bErr := FALSE;
      Busy := TRUE;
   END_IF
END_IF

IF bStarted THEN
   (* raising edge of Timer triggers write request *)
   fbWrite( NetID := '', Port := 553, IdxGrp := nIdxGrp, IdxOffs := 16#00000049,
         LEN := 2, SrcAddr := ADR(nType), WRITE := bStarted, TMOUT := T#1s);
   IF NOT fbWrite.Busy THEN
      (* There was an error in the execution of the write request *)
      IF fbWrite.Err THEN
         bErr := TRUE;
      END_IF
      fbWrite(WRITE := FALSE);    (* reset because of edge detection in FB ADSWRITE *)
      bStarted := FALSE;
      Busy := FALSE;
   END_IF
END_IF

END_FUNCTION_BLOCK

// CNC/6 BlockSearch/ReadBsType
FUNCTION_BLOCK ReadBsType
VAR_INPUT
	nIdxGrp: UDINT;
	bStart: BOOL;
	pDest: POINTER TO UINT;
END_VAR
VAR_OUTPUT
	Busy: BOOL;
	bErr: BOOL;
END_VAR
VAR
	fbRead: ADSREAD;
	bStarted: BOOL;
END_VAR

IF bStarted = FALSE THEN
   IF bStart = TRUE THEN
      bStarted := TRUE;
      bErr := FALSE;
      Busy := TRUE;
   END_IF
END_IF

IF bStarted THEN
   (* raising edge of Timer triggers read request *)
   fbRead( NetID := '', Port := 553, IdxGrp := nIdxGrp, IdxOffs := 16#00000061,
         LEN := 2, DestAddr := pDest, READ := bStarted, TMOUT := T#1s);
   IF NOT fbRead.Busy THEN
      (* There was an error in the execution of the read request *)
      IF fbRead.Err THEN
         bErr := TRUE;
      END_IF
      fbRead(READ := FALSE);    (* reset because of edge detection in FB ADSREAD *)
      bStarted := FALSE;
      Busy := FALSE;
   END_IF
END_IF

END_FUNCTION_BLOCK

// CNC/6 BlockSearch/WriteBsCoveredDistance
FUNCTION_BLOCK WriteBsCoveredDistance
VAR_INPUT
	nIdxGrp: UDINT;
	bStart: BOOL;
	fDistance: LREAL;
END_VAR
VAR_OUTPUT
	Busy: BOOL;
	bErr: BOOL;
END_VAR
VAR
	fbWrite: ADSWRITE;
	bStarted: BOOL;
END_VAR

IF bStarted = FALSE THEN
   IF bStart = TRUE THEN
      bStarted := TRUE;
      bErr := FALSE;
      Busy := TRUE;
   END_IF
END_IF

IF bStarted THEN
   (* raising edge of Timer triggers write request *)
   fbWrite( NetID := '', Port := 553, IdxGrp := nIdxGrp, IdxOffs := 16#0000004A,
         LEN := 8, SrcAddr := ADR(fDistance), WRITE := bStarted, TMOUT := T#1s);
   IF NOT fbWrite.Busy THEN
      (* There was an error in the execution of the write request *)
      IF fbWrite.Err THEN
         bErr := TRUE;
      END_IF
      fbWrite(WRITE := FALSE);    (* reset because of edge detection in FB ADSWRITE *)
      bStarted := FALSE;
      Busy := FALSE;
   END_IF
END_IF

END_FUNCTION_BLOCK

// CNC/6 BlockSearch/ReadBsCoveredDistance
FUNCTION_BLOCK ReadBsCoveredDistance
VAR_INPUT
	nIdxGrp: UDINT;
	bStart: BOOL;
	pDest: POINTER TO LREAL;
END_VAR
VAR_OUTPUT
	Busy: BOOL;
	bErr: BOOL;
END_VAR
VAR
	fbRead: ADSREAD;
	bStarted: BOOL;
END_VAR

IF bStarted = FALSE THEN
   IF bStart = TRUE THEN
      bStarted := TRUE;
      bErr := FALSE;
      Busy := TRUE;
   END_IF
END_IF

IF bStarted THEN
   (* raising edge of Timer triggers read request *)
   fbRead( NetID := '', Port := 553, IdxGrp := nIdxGrp, IdxOffs := 16#00000062,
         LEN := 8, DestAddr := pDest, READ := bStarted, TMOUT := T#1s);
   IF NOT fbRead.Busy THEN
      (* There was an error in the execution of the read request *)
      IF fbRead.Err THEN
         bErr := TRUE;
      END_IF
      fbRead(READ := FALSE);    (* reset because of edge detection in FB ADSREAD *)
      bStarted := FALSE;
      Busy := FALSE;
   END_IF
END_IF

END_FUNCTION_BLOCK

// CNC/6 BlockSearch/WriteBsAutoReturn
FUNCTION_BLOCK WriteBsAutoReturn
VAR_INPUT
	nIdxGrp: UDINT;
	bStart: BOOL;
	bAutoReturn: BOOL;
END_VAR
VAR_OUTPUT
	Busy: BOOL;
	bErr: BOOL;
END_VAR
VAR
	fbWrite: ADSWRITE;
	bStarted: BOOL;
END_VAR

IF bStarted = FALSE THEN
   IF bStart = TRUE THEN
      bStarted := TRUE;
      bErr := FALSE;
      Busy := TRUE;
   END_IF
END_IF

IF bStarted THEN
   (* raising edge of Timer triggers write request *)
   fbWrite( NetID := '', Port := 553, IdxGrp := nIdxGrp, IdxOffs := 16#0000004B,
         LEN := 1, SrcAddr := ADR(bAutoReturn), WRITE := bStarted, TMOUT := T#1s);
   IF NOT fbWrite.Busy THEN
      (* There was an error in the execution of the write request *)
      IF fbWrite.Err THEN
         bErr := TRUE;
      END_IF
      fbWrite(WRITE := FALSE);    (* reset because of edge detection in FB ADSWRITE *)
      bStarted := FALSE;
      Busy := FALSE;
   END_IF
END_IF

END_FUNCTION_BLOCK

// CNC/6 BlockSearch/ReadBsAutoReturn
FUNCTION_BLOCK ReadBsAutoReturn
VAR_INPUT
	nIdxGrp: UDINT;
	bStart: BOOL;
	pDest: POINTER TO BOOL;
END_VAR
VAR_OUTPUT
	Busy: BOOL;
	bErr: BOOL;
END_VAR
VAR
	fbRead: ADSREAD;
	bStarted: BOOL;
END_VAR

IF bStarted = FALSE THEN
   IF bStart = TRUE THEN
      bStarted := TRUE;
      bErr := FALSE;
      Busy := TRUE;
   END_IF
END_IF

IF bStarted THEN
   (* raising edge of Timer triggers read request *)
   fbRead( NetID := '', Port := 553, IdxGrp := nIdxGrp, IdxOffs := 16#00000063,
         LEN := 1, DestAddr := pDest, READ := bStarted, TMOUT := T#1s);
   IF NOT fbRead.Busy THEN
      (* There was an error in the execution of the read request *)
      IF fbRead.Err THEN
         bErr := TRUE;
      END_IF
      fbRead(READ := FALSE);    (* reset because of edge detection in FB ADSREAD *)
      bStarted := FALSE;
      Busy := FALSE;
   END_IF
END_IF

END_FUNCTION_BLOCK

// CNC/6 BlockSearch/WriteBsDeviationMax
FUNCTION_BLOCK WriteBsDeviationMax
VAR_INPUT
	nIdxGrp: UDINT;
	bStart: BOOL;
	nDeviationMax: UDINT;
END_VAR
VAR_OUTPUT
	Busy: BOOL;
	bErr: BOOL;
END_VAR
VAR
	fbWrite: ADSWRITE;
	bStarted: BOOL;
END_VAR

IF bStarted = FALSE THEN
   IF bStart = TRUE THEN
      bStarted := TRUE;
      bErr := FALSE;
      Busy := TRUE;
   END_IF
END_IF

IF bStarted THEN
   (* raising edge of Timer triggers write request *)
   fbWrite( NetID := '', Port := 553, IdxGrp := nIdxGrp, IdxOffs := 16#0000004C,
         LEN := 4, SrcAddr := ADR(nDeviationMax), WRITE := bStarted, TMOUT := T#1s);
   IF NOT fbWrite.Busy THEN
      (* There was an error in the execution of the write request *)
      IF fbWrite.Err THEN
         bErr := TRUE;
      END_IF
      fbWrite(WRITE := FALSE);    (* reset because of edge detection in FB ADSWRITE *)
      bStarted := FALSE;
      Busy := FALSE;
   END_IF
END_IF

END_FUNCTION_BLOCK

// CNC/6 BlockSearch/ReadBsDeviationMax
FUNCTION_BLOCK ReadBsDeviationMax
VAR_INPUT
	nIdxGrp: UDINT;
	bStart: BOOL;
	pDest: POINTER TO UDINT;
END_VAR
VAR_OUTPUT
	Busy: BOOL;
	bErr: BOOL;
END_VAR
VAR
	fbRead: ADSREAD;
	bStarted: BOOL;
END_VAR

IF bStarted = FALSE THEN
   IF bStart = TRUE THEN
      bStarted := TRUE;
      bErr := FALSE;
      Busy := TRUE;
   END_IF
END_IF

IF bStarted THEN
   (* raising edge of Timer triggers read request *)
   fbRead( NetID := '', Port := 553, IdxGrp := nIdxGrp, IdxOffs := 16#00000064,
         LEN := 4, DestAddr := pDest, READ := bStarted, TMOUT := T#1s);
   IF NOT fbRead.Busy THEN
      (* There was an error in the execution of the read request *)
      IF fbRead.Err THEN
         bErr := TRUE;
      END_IF
      fbRead(READ := FALSE);    (* reset because of edge detection in FB ADSREAD *)
      bStarted := FALSE;
      Busy := FALSE;
   END_IF
END_IF

END_FUNCTION_BLOCK

// CNC/6 BlockSearch/WriteBsBlockNumber
FUNCTION_BLOCK WriteBsBlockNumber
VAR_INPUT
	nIdxGrp: UDINT;
	bStart: BOOL;
	nBlockNumber: DINT;
END_VAR
VAR_OUTPUT
	Busy: BOOL;
	bErr: BOOL;
END_VAR
VAR
	fbWrite: ADSWRITE;
	bStarted: BOOL;
END_VAR

IF bStarted = FALSE THEN
   IF bStart = TRUE THEN
      bStarted := TRUE;
      bErr := FALSE;
      Busy := TRUE;
   END_IF
END_IF

IF bStarted THEN
   (* raising edge of Timer triggers write request *)
   fbWrite( NetID := '', Port := 553, IdxGrp := nIdxGrp, IdxOffs := 16#0000005F,
         LEN := 4, SrcAddr := ADR(nBlockNumber), WRITE := bStarted, TMOUT := T#1s);
   IF NOT fbWrite.Busy THEN
      (* There was an error in the execution of the write request *)
      IF fbWrite.Err THEN
         bErr := TRUE;
      END_IF
      fbWrite(WRITE := FALSE);    (* reset because of edge detection in FB ADSWRITE *)
      bStarted := FALSE;
      Busy := FALSE;
   END_IF
END_IF

END_FUNCTION_BLOCK

// CNC/6 BlockSearch/ReadBsBlockNumber
FUNCTION_BLOCK ReadBsBlockNumber
VAR_INPUT
	nIdxGrp: UDINT;
	bStart: BOOL;
	pDest: POINTER TO DINT;
END_VAR
VAR_OUTPUT
	Busy: BOOL;
	bErr: BOOL;
END_VAR
VAR
	fbRead: ADSREAD;
	bStarted: BOOL;
END_VAR

IF bStarted = FALSE THEN
   IF bStart = TRUE THEN
      bStarted := TRUE;
      bErr := FALSE;
      Busy := TRUE;
   END_IF
END_IF

IF bStarted THEN
   (* raising edge of Timer triggers read request *)
   fbRead( NetID := '', Port := 553, IdxGrp := nIdxGrp, IdxOffs := 16#00000077,
         LEN := 4, DestAddr := pDest, READ := bStarted, TMOUT := T#1s);
   IF NOT fbRead.Busy THEN
      (* There was an error in the execution of the read request *)
      IF fbRead.Err THEN
         bErr := TRUE;
      END_IF
      fbRead(READ := FALSE);    (* reset because of edge detection in FB ADSREAD *)
      bStarted := FALSE;
      Busy := FALSE;
   END_IF
END_IF

END_FUNCTION_BLOCK

// CNC/6 BlockSearch/WriteBsBlockCount
FUNCTION_BLOCK WriteBsBlockCount
VAR_INPUT
	nIdxGrp: UDINT;
	bStart: BOOL;
	nBlockCount: DINT;
END_VAR
VAR_OUTPUT
	Busy: BOOL;
	bErr: BOOL;
END_VAR
VAR
	fbWrite: ADSWRITE;
	bStarted: BOOL;
END_VAR

IF bStarted = FALSE THEN
   IF bStart = TRUE THEN
      bStarted := TRUE;
      bErr := FALSE;
      Busy := TRUE;
   END_IF
END_IF

IF bStarted THEN
   (* raising edge of Timer triggers write request *)
   fbWrite( NetID := '', Port := 553, IdxGrp := nIdxGrp, IdxOffs := 16#0000005E,
         LEN := 4, SrcAddr := ADR(nBlockCount), WRITE := bStarted, TMOUT := T#1s);
   IF NOT fbWrite.Busy THEN
      (* There was an error in the execution of the write request *)
      IF fbWrite.Err THEN
         bErr := TRUE;
      END_IF
      fbWrite(WRITE := FALSE);    (* reset because of edge detection in FB ADSWRITE *)
      bStarted := FALSE;
      Busy := FALSE;
   END_IF
END_IF

END_FUNCTION_BLOCK

// CNC/6 BlockSearch/ReadBsBlockCount
FUNCTION_BLOCK ReadBsBlockCount
VAR_INPUT
	nIdxGrp: UDINT;
	bStart: BOOL;
	pDest: POINTER TO DINT;
END_VAR
VAR_OUTPUT
	Busy: BOOL;
	bErr: BOOL;
END_VAR
VAR
	fbRead: ADSREAD;
	bStarted: BOOL;
END_VAR

IF bStarted = FALSE THEN
   IF bStart = TRUE THEN
      bStarted := TRUE;
      bErr := FALSE;
      Busy := TRUE;
   END_IF
END_IF

IF bStarted THEN
   (* raising edge of Timer triggers read request *)
   fbRead( NetID := '', Port := 553, IdxGrp := nIdxGrp, IdxOffs := 16#00000076,
         LEN := 4, DestAddr := pDest, READ := bStarted, TMOUT := T#1s);
   IF NOT fbRead.Busy THEN
      (* There was an error in the execution of the read request *)
      IF fbRead.Err THEN
         bErr := TRUE;
      END_IF
      fbRead(READ := FALSE);    (* reset because of edge detection in FB ADSREAD *)
      bStarted := FALSE;
      Busy := FALSE;
   END_IF
END_IF

END_FUNCTION_BLOCK

// CNC/6 BlockSearch/WriteBsPass
FUNCTION_BLOCK WriteBsPass
VAR_INPUT
	nIdxGrp: UDINT;
	bStart: BOOL;
	nPass: DINT;
END_VAR
VAR_OUTPUT
	Busy: BOOL;
	bErr: BOOL;
END_VAR
VAR
	fbWrite: ADSWRITE;
	bStarted: BOOL;
END_VAR

IF bStarted = FALSE THEN
   IF bStart = TRUE THEN
      bStarted := TRUE;
      bErr := FALSE;
      Busy := TRUE;
   END_IF
END_IF

IF bStarted THEN
   (* raising edge of Timer triggers write request *)
   fbWrite( NetID := '', Port := 553, IdxGrp := nIdxGrp, IdxOffs := 16#00000060,
         LEN := 4, SrcAddr := ADR(nPass), WRITE := bStarted, TMOUT := T#1s);
   IF NOT fbWrite.Busy THEN
      (* There was an error in the execution of the write request *)
      IF fbWrite.Err THEN
         bErr := TRUE;
      END_IF
      fbWrite(WRITE := FALSE);    (* reset because of edge detection in FB ADSWRITE *)
      bStarted := FALSE;
      Busy := FALSE;
   END_IF
END_IF

END_FUNCTION_BLOCK

// CNC/6 BlockSearch/ReadBsPass
FUNCTION_BLOCK ReadBsPass
VAR_INPUT
	nIdxGrp: UDINT;
	bStart: BOOL;
	pDest: POINTER TO DINT;
END_VAR
VAR_OUTPUT
	Busy: BOOL;
	bErr: BOOL;
END_VAR
VAR
	fbRead: ADSREAD;
	bStarted: BOOL;
END_VAR

IF bStarted = FALSE THEN
   IF bStart = TRUE THEN
      bStarted := TRUE;
      bErr := FALSE;
      Busy := TRUE;
   END_IF
END_IF

IF bStarted THEN
   (* raising edge of Timer triggers read request *)
   fbRead( NetID := '', Port := 553, IdxGrp := nIdxGrp, IdxOffs := 16#00000078,
         LEN := 4, DestAddr := pDest, READ := bStarted, TMOUT := T#1s);
   IF NOT fbRead.Busy THEN
      (* There was an error in the execution of the read request *)
      IF fbRead.Err THEN
         bErr := TRUE;
      END_IF
      fbRead(READ := FALSE);    (* reset because of edge detection in FB ADSREAD *)
      bStarted := FALSE;
      Busy := FALSE;
   END_IF
END_IF

END_FUNCTION_BLOCK

// CNC/8 Mis/FB_WriteCNCZeroOffset
/// ------------------------------------------------------------------------------------ 
/// Desc:	Description																	
///**************************************************************************************
///**************************************************************************************
///	 Write NPV Value directly to CNC core using V.G. Variables via ADS	
///**************************************************************************************
FUNCTION_BLOCK FB_WriteCNCZeroOffset
VAR_INPUT
	/// rising edge to start 
	bExecute: BOOL;
	/// which table, G54=1, G55=2, G55=3, .... 
	nG159Index: BYTE;
	/// Channel Indedx
	nChanIdx: UDINT;
	/// Axis name in channel 
	sAxisName: STRING(95);
	/// value to set 
	lrValue: LREAL;
END_VAR
VAR_OUTPUT
	bBusy: BOOL;
	bError: BOOL;
	nErrorID: UDINT;
END_VAR
VAR
	fbAdsWrite: ADSWRITE;
	stCNCG159VG: ST_CNCG159VG;
END_VAR

stCNCG159VG.dValue := LREAL_TO_DINT(lrValue * 10000);
stCNCG159VG.sTarget := 'V.G.NP[';
stCNCG159VG.sTarget := CONCAT(stCNCG159VG.sTarget, BYTE_TO_STRING(nG159Index));
stCNCG159VG.sTarget := CONCAT(stCNCG159VG.sTarget, '].V.');
stCNCG159VG.sTarget := CONCAT(stCNCG159VG.sTarget,sAxisName);

fbAdsWrite(
	PORT:= 552 ,
	IDXGRP:= 16#22300 + nChanIdx+1,
	IDXOFFS:=16#3F,
	LEN:= SIZEOF(stCNCG159VG) ,
	SRCADDR:=ADR(stCNCG159VG) ,
	WRITE:= bExecute,
	TMOUT:= ,
	BUSY=> bBusy,
	ERR=> bError ,
	ERRID=> nErrorID);

END_FUNCTION_BLOCK

// CNC/8 Mis/FB_WriteCNCZeroOffsetDefault
/// ------------------------------------------------------------------------------------ 
/// Desc:	Description																	
///**************************************************************************************
///**************************************************************************************
///	 Write NPV Default (the active table afetr reset) directly to CNC core using V.G. Variables via ADS	
///**************************************************************************************
FUNCTION_BLOCK FB_WriteCNCZeroOffsetDefault
VAR_INPUT
	/// rising edge to start 
	bExecute: BOOL;
	/// which table, G54=1, G55=2, G55=3, .... 
	nG159Index: BYTE;
	/// Channel Indedx
	nChanIdx: UDINT;
END_VAR
VAR_OUTPUT
	bBusy: BOOL;
	bError: BOOL;
	nErrorID: UDINT;
END_VAR
VAR
	fbAdsWrite: ADSWRITE;
	stCNCG159VG: ST_CNCG159VG;
END_VAR

stCNCG159VG.dValue := nG159Index;
stCNCG159VG.sTarget := 'V.G.NP_DEFAULT';

fbAdsWrite(
	PORT:= 552 ,
	IDXGRP:= 16#22300 + nChanIdx+1,
	IDXOFFS:=16#3F,
	LEN:= SIZEOF(stCNCG159VG) ,
	SRCADDR:=ADR(stCNCG159VG) ,
	WRITE:= bExecute,
	TMOUT:= ,
	BUSY=> bBusy,
	ERR=> bError ,
	ERRID=> nErrorID);

END_FUNCTION_BLOCK

// CNC/8 Mis/HLI_HandleMessages
FUNCTION_BLOCK HLI_HandleMessages
VAR_INPUT
	/// Enable 
	bEnable: BOOL;
	/// Number of channel 
	nChanIdx: INT;
	/// Channelstruct 
	pChannel: POINTER TO ST_CncChannel;
END_VAR
VAR_OUTPUT
	bNewMessage: BOOL;
	bError: BOOL;
	sMessage: STRING(255);
END_VAR
VAR
	/// Index of channel specific HLI area 

	bFirstCycle: BOOL := TRUE;
	bModeChanged: BOOL;
	nState: USINT;
	nActMode: UDINT;
	dwCncState: DWORD;
	fbRtrigStateStart: R_TRIG;
	pString: POINTER TO STRING(HLI_MSG_CONTENT_STRL);
	fbLog: ADSLOGEVENT;
	stMessageData: TcEvent;
END_VAR
VAR CONSTANT
	sFormat: STRING(2) := '%s';
END_VAR

(******************************************************************************)
(* Name:		HLI_HandleMessages											 	*)
(* Date:		08/12/01													 	*)
(* Author:	H. Rausch (Beckhoff Automation GmbH)							 	*)
(* Ver:		1.0																	*)
(* Desc:		Function block for recieving messages from CNC and passing them to*)
(*				the TwinCAT EventLogger. Only the latest message from CNC is 	*)
(*				active there. The event will be resetted if a new message from	*)
(*				CNC is recieved, the CNC state changes to 'ACTIVE', the CNC mode*)
(*				is changed or the channel is resetted							*)
(*																				*)
(*				Messages are passed as a fill string to the event logger with 	*)
(*				source id 9000 and event id 1. This requires a correspondant 	*)
(*				configuration in the tceventsourcelocation.xml and in an		*)
(*				associated message file!										*)
(* ---------------------------------------------------------------------------*)
(* Rev:		Add new version number here!										*)
(* Date.		Add revision data here											*)
(* Desc:		Add revision description here!									*)
(******************************************************************************)

(* Write event config data once on start up *)
IF bFirstCycle THEN
	stMessageData.bQuitRequired			:= TRUE;
	stMessageData.Class					:= TCEVENTCLASS_MESSAGE;
	stMessageData.DataFormatStrAddress	:= ADR(sFormat);
	stMessageData.Prio					:= 0;
	stMessageData.Id					:= 1;
	stMessageData.SourceId 				:= 9000;
	stMessageData.Flags 				:= TCEVENTFLAG_LOG OR TCEVENTFLAG_SRCID;
	stMessageData.StreamType			:= TCEVENTSTREAM_SIMPLE;
	stMessageData.ProgId 				:= 'TcEventFormatter.TcXmlFormatter';
END_IF



(* Check for zero pointer and leave fb if necessary *)
IF NOT HLI3_CheckChannelValid(nChannel := nChanIdx) THEN
	RETURN;
END_IF
	(* Check CNC state *)
	dwCncState := HLI3_GetChannelState(nChanIdx:=nChanIdx);

	(* Rising trig if CNC state changes to ACTIVE *)
	fbRtrigStateStart
		(CLK := (dwCncState = HLI_IMCM_PROCESS_ACTIVE));

	(* Watch CNC mode *)
	bModeChanged	:= (nActMode <> pChannel^.ActMode);
	nActMode 		:= pChannel^.ActMode;

IF NOT bEnable THEN
	gpCh[nChanIdx]^.msg_mc_control.enable_w				:= FALSE;
	gpCh[nChanIdx]^.msg_mc_control.request_semaphor_rw	:= FALSE;
	sMessage										:= '';
ELSE
	gpCh[nChanIdx]^.msg_mc_control.enable_w 			:= TRUE;

	CASE nState OF
	 0:
		(* Wait for new messages from CNC *)
		IF gpCh[nChanIdx]^.msg_mc_control.request_semaphor_rw THEN
			(* Convert byte stream to string *)
			pString  := ADR(gpCh[nChanIdx]^.msg_mc_control.request_r.inhalt);
			sMessage := pString^;
			(* Reset notification from HLI *)
			gpCh[nChanIdx]^.msg_mc_control.request_semaphor_rw := FALSE;

			nState := 1;
		END_IF

	 1:
		(* Wait that ADSEVENTLOG instance is cleared *)
		IF (fbLog.EventState = 0) THEN
			nState := 2;
		END_IF

	 2:
		(* Set message to eventlogger *)
		IF (fbLog.EventState > 0) THEN
			nState := 0;
		END_IF

	END_CASE

	(* Managing Eventlogger *)
	fbLog
		(NETID				:= '',
		 PORT					:= 110,
		 Event				:= (nState = 2),
		 EventQuit			:= (nState = 1) OR
									(dwCncState = HLI_IMCM_PROCESS_RESETTING) OR
									fbRtrigStateStart.Q OR
									bModeChanged,
		 EventConfigData	:= stMessageData,
		 EventDataAddress	:= ADR(sMessage),
		 EventDataLength	:= SIZEOF(sMessage),
		 TMOUT				:= t#2s
		);
END_IF

(* Reset first cycle indicator *)
bFirstCycle := FALSE;

END_FUNCTION_BLOCK

// CNC/8 Mis/HLI_MoveSpindle
///*********************************************************************************************************
///NAME.......................:	HLI_MoveSpindle	
///DATUM....................:	7.9.2009
///AUTOR....................:	Michael Balsfulland (MiB)
///VERSION................:	1.2
///				1.1 20.8.2010 MiB: kompletter Umbau auf Schrittkette mit Fehlerhandling
///				1.2 15.08.2017 MiB: BugFix: Linkslauf: Vorgabe der Drehzahl muss positiv erfolgen 
///BESCHREIBUNG.:	 Spindel mit einer vorgegeben Geschwindigkeit starten oder Spindel stoppen
///......................: 	
///
///**********************************************************************************************************
FUNCTION_BLOCK HLI_MoveSpindle
VAR
	pUnit: POINTER TO MC_CONTROL_EXT_TO_IPO;
	fbRTrigStart: R_TRIG;
	fbRTrigStop: R_TRIG;
	nState: INT;
	/// Index of axis specific HLI area 
	nHliAxIfcIdx: UDINT;
END_VAR
VAR_INPUT
	/// Spindel Achssnummer 
	nLogAxisNr: UDINT;
	/// U/min 
	nSpeed: DINT;
	/// steigende Flanke 
	bStart: BOOL;
	/// steigende Flanke 
	bStop: BOOL;
END_VAR
VAR_OUTPUT
	bBusy: BOOL;
	bError: BOOL;
	nErrID: INT;
	sErrText: STRING;
END_VAR

fbRTrigStart(clk := bStart);
IF fbRTrigStart.Q THEN
	bError := FALSE;
	nErrId := 0;
	sErrText := '';
	nState := 100;   (* Spindel starten *)
END_IF


fbRTrigStop(clk := bStop);
IF fbRTrigStop.Q THEN
	bError := FALSE;
	nErrId := 0;
	sErrText := '';
	nState := 200;  (* Spindel stoppen *)
END_IF

nHliAxIfcIdx := nLogAxisNr - 1;

IF fbRTrigStop.Q OR fbRTrigStart.Q THEN   (* Grundzustände testen *)
	bBusy := TRUE;
	IF nLogAxisNr = 0 THEN
		nState := -1;
		nErrID := 1;
		sErrText := 'Spindel ID = 0';
	END_IF
	IF ADR(gpAx[nHliAxIfcIdx]^)  = 0  THEN
		nState := -1;
		nErrID := 2;
		sErrText := 'Achsstruktur nicht vorhanden -> eventuell HLI Init nicht OK';
	END_IF
	IF gpAx[nHliAxIfcIdx]^.ipo_state.spindle_axis_r <> TRUE THEN
		nState := -1;
		nErrID := 3;
		sErrText := 'Achse ist kene Spindel';
	END_IF
END_IF

CASE nState OF


-1: (* Fehler *)
   	bError := TRUE;
	bBusy := FALSE;

0: (* IDLE *)
	bBusy := FALSE;


100: (* Spindel starten *)
	(* Check Override *)
	gpAx[nHliAxIfcIdx]^.ipo_mc_control.override.enable_w := TRUE;
	IF gpAx[nHliAxIfcIdx]^.ipo_mc_control.override.state_r = 0 THEN
		nState := -1;
		nErrID := 4;
		sErrText := 'Spindeloverride = 0';
	ELSE
		nState := 110;
	END_IF


110: (* Parametrieren des Aufrufs *)
	pUnit := ADR(gpAx[nHliAxIfcIdx]^.ipo_mc_control.ext_to_ipo);
	IF (nSpeed > 0) THEN
		pUnit^.command_w.vb_prog   :=  nSpeed * 360 / 60 * 1000  ;(*Programmierter Satzvorschub in u/min*)
		pUnit^.command_w.dreh_info := 1;(* rechtslauf *)
	ELSE
		pUnit^.command_w.vb_prog   :=  -nSpeed * 360 / 60 * 1000  ;(*Programmierter Satzvorschub in u/min*)
		pUnit^.command_w.dreh_info := 0;(* linkslauf*)
	END_IF
	pUnit^.command_w.geo_gm_fkt    := 0;(*G- und M- Fkt.-Bitleiste*)
	pUnit^.command_w.satz_typ      := HLI_NC_MOVE_ENDLOS;(*Einer der Werte: HLI_NC_MOVE_LIN, HLI_NC_MOVREF, HLI_NC_MOVE_ENDLOS, HLI_NC_SPINDEL_STOP*)
	IF pUnit^.command_semaphor_rw = FALSE THEN
	    pUnit^.command_semaphor_rw := TRUE;
	    nState := 120;
	END_IF

	IF (nSpeed=0) THEN
		nState := -1;
		nErrID := 6;
		sErrText := 'Vorgabegeschwindigkeit = 0';
	END_IF

120: (* Start *)

	IF pUnit^.command_semaphor_rw = FALSE THEN
	    nState := 300;  (* checken Auftragsfehler *)
	END_IF



200: (* Spindel Stopp*)
	pUnit := ADR(gpAx[nHliAxIfcIdx]^.ipo_mc_control.ext_to_ipo);
	pUnit^.command_w.satz_typ  := HLI_NC_SPINDEL_STOP;(*Einer der Werte: HLI_NC_MOVE_LIN, HLI_NC_MOVREF, HLI_NC_MOVE_ENDLOS, HLI_NC_SPINDEL_STOP*)
	pUnit^.command_w.dreh_info := 0;(*Drehinformation*)
	IF pUnit^.command_semaphor_rw = FALSE THEN
	    pUnit^.command_semaphor_rw := TRUE;
	    nState := 210;
	END_IF

210: (* Warten auf Stop *)
	IF pUnit^.command_semaphor_rw = FALSE THEN
	    nState := 300;   (* checken Auftragsfehler *)
	END_IF

300: (* checken Auftragsfehler *)
	IF (gpAx[nHliAxIfcIdx]^.ipo_state.spindle_order_error_r) THEN
		nState := -1;
		nErrID := 5;
		sErrText := 'Beauftragunsfehler Spindel';
	ELSE
		nState := 310;
	END_IF

310: (* Warten auf Solldrehzahl erreicht *)

	IF (gpAx[nHliAxIfcIdx]^.lr_state.rev_erreicht_r) THEN
		nState := 0;
	END_IF


END_CASE


(*
IF nLogAxisNr <> 0 THEN
	IF pAC[nLogAxisNr] <> 0  THEN
		IF ADR(gpAx[nLogAxisNr]^) <> 0  THEN
			IF gpAx[nLogAxisNr]^.ipo_state.X_SpindleAxis = TRUE THEN

				(* command spindle revolution *)
				IF fbRTrigStart.Q THEN
					pCommand := ADR(gpAx[nLogAxisNr]^.ipo_mc_control.MCControlExtToIpo_ExtToIpo);
					IF (nSpeed > 0) THEN
						pCommand^.command_w.D_VbProg :=  DINT_TO_UDINT((nSpeed * 360 / 60) * 1000)  ;(*Programmierter Satzvorschub in u/min*)
  						pCommand^.command_w.W_DrehInfo := 1;(* rechtslauf *)
					ELSE
						pCommand^.command_w.D_VbProg :=  DINT_TO_UDINT((-nSpeed * 360 / 60) * 1000)  ;(*Programmierter Satzvorschub in u/min*)
						pCommand^.command_w.W_DrehInfo := 0;(* linkslauf*)
					END_IF
					pCommand^.command_w.D_GeoGmFkt := 0;(*G- und M- Fkt.-Bitleiste*)
					pCommand^.command_w.W_SatzTyp := HLI_NC_MOVE_ENDLOS;(*Einer der Werte: HLI_NC_MOVE_LIN, HLI_NC_MOVREF, HLI_NC_MOVE_ENDLOS, HLI_NC_SPINDEL_STOP*)
					pCommand^.command_semaphor_rw := TRUE;
				END_IF
				(* command spindle revolution *)
				IF fbRTrigStop.Q THEN
					pCommand := ADR(gpAx[nLogAxisNr]^.ipo_mc_control.MCControlExtToIpo_ExtToIpo);
					pCommand^.command_w.D_VbProg := 600000000;(*Programmierter Satzvorschub*)
					pCommand^.command_w.D_GeoGmFkt := 0;(*G- und M- Fkt.-Bitleiste*)

					pCommand^.command_w.W_SatzTyp := HLI_NC_SPINDEL_STOP;(*Einer der Werte: HLI_NC_MOVE_LIN, HLI_NC_MOVREF, HLI_NC_MOVE_ENDLOS, HLI_NC_SPINDEL_STOP*)
					pCommand^.command_w.W_DrehInfo := 0;(*Drehinformation*)
					pCommand^.command_semaphor_rw := TRUE;
				END_IF
			END_IF
		END_IF
	END_IF
END_IF
*)

END_FUNCTION_BLOCK

// CNC/8 Mis/HLI3_CheckCNCAlive
PROGRAM HLI3_CheckCNCAlive
VAR_INPUT
	nChanIdx: INT;
END_VAR

VAR
	bMessageDisplayed : BOOL;
END_VAR

(* The assumption is made that the cycle time of the PLC is at least twice as big as the CNC cycle time.

The Cycle time of CNC is displayed in element:
	pMC[1]^.addr^.HLIHeadChannel_Data.LCWatchDogUnit_lc.D_cycle_time_r

remark: Take care if PLC cycle is smaller not to check CNC faster as possible !!!

To simulate failure of CNC set cycle time of PLC smaller than CNC (Resource/task configuration).
*)

// HLI3_CheckCNCAlive := FALSE;
IF NOT HLI3_CheckChannelValid(nChannel := nChanIdx) THEN
	RETURN;
END_IF
 
(* Copy current state of live sign to watchdog state    *)
gpCh[nChanIdx]^.head.lc_watchdog.alive_rw
	:= gpCh[nChanIdx]^.head.lc_watchdog.alive_rw;

IF gpCh[nChanIdx]^.head.lc_watchdog.alive_rw = FALSE AND NOT bMessageDisplayed THEN
	(* PLC detects CNC not alive -> start individual emergency stop within PLC *)
	ADSLOGSTR( msgCtrlMask := ADSLOG_MSGTYPE_ERROR OR
							ADSLOG_MSGTYPE_MSGBOX OR
							ADSLOG_MSGTYPE_LOG,
			msgFmtStr := 'PLC detects CNC not alive: %s',
			strArg := 'channel 1');
			
			bMessageDisplayed := TRUE;
END_IF


(* assign return value *)
//HLI3_CheckCNCAlive := gpCh[nChanIdx]^.head.lc_watchdog.alive_rw;

(* reset live sign for next cycle *)
gpCh[nChanIdx]^.head.lc_watchdog.alive_rw := FALSE;

END_PROGRAM

// CNC/8 Mis/HLI3_GetLogAxisId
FUNCTION HLI3_GetLogAxisId : INT
VAR_INPUT
	nHliAxisIdx: INT;
END_VAR
VAR
	i: INT;
END_VAR

(* ========================================================= *)
(*    FUN: HLI3_GetLogAxisId                            	 *)
(* --------------------------------------------------------- *)
(*   Desc: returns the Log. Axis Idx for a given HLI Index   *)
(*   Author: TV                                              *)
(*   Date: 22.01.2014                                        *)
(*   Rev.: 1.0                                               *)
(* ========================================================= *)
HLI3_GetLogAxisId := -1;
IF NOT HLI3_CheckAxisValid(nHliAxisIdx := nHliAxisIdx) THEN
	RETURN;
END_IF

HLI3_GetLogAxisId := UINT_TO_INT(gpAx[nHliAxisIdx]^.head.log_ax_nr_r);

END_FUNCTION

// CNC/8 Mis/HLI3_ResetSpindle
FUNCTION HLI3_ResetSpindle : BOOL
VAR_INPUT
	/// axis number of spindle 
	nHliAxisIdx: INT;
END_VAR
VAR
	/// Index of axis specific HLI area 
	nHliAxIfcIdx: INT;
	SpdlState: BOOL;
	SpdlCommand: BOOL;
	ResetCmd: BOOL := FALSE;
	/// local pointer to data of actual axis 
	pResetUnit: POINTER TO MC_CONTROL_BOOL_UNIT;
END_VAR

HLI3_ResetSpindle := FALSE;

IF NOT HLI3_CheckAxisValid(nHliAxisIdx := nHliAxisIdx) THEN
	HLI3_ResetSpindle := FALSE;
	RETURN;
END_IF

	pResetUnit := ADR(gpAx[nHliAxisIdx]^.ipo_mc_control.spdl_reset);
	SpdlState  := pResetUnit^.state_r;

	IF ResetCmd = TRUE THEN
		pResetUnit^.command_w := TRUE;
		SpdlCommand           := pResetUnit^.command_w;
		HLI3_ResetSpindle          := SpdlState;
	END_IF

END_FUNCTION

// CNC/8 Mis/HLI3_SetPLCAlive
FUNCTION HLI3_SetPLCAlive : BOOL
VAR_INPUT
	nChanIdx: INT;
END_VAR

(*
Display PLC is just alive (Trigger Watchdog to MC)
If PLC is stopped here, alive sign is missing.
-> CNC raises error message
-> CNC stoppes movement with internal FEEDHOLD
-> system has to be restarted (after removal of error)
*)

HLI3_SetPLCAlive := FALSE;
IF NOT HLI3_CheckChannelValid(nChannel := nChanIdx) THEN
	RETURN;
END_IF
gpCh[nChanIdx]^.head.mc_watchdog.cycle_time_w := 2000;   // Watchdog time 2000 µs
gpCh[nChanIdx]^.head.mc_watchdog.enable_w := TRUE;
gpCh[nChanIdx]^.head.mc_watchdog.alive_rw := TRUE;

HLI3_SetPLCAlive := TRUE;

END_FUNCTION

// CNC/8 Mis/PB_10_CNC_Spindelkopplung
PROGRAM PB_10_CNC_Spindelkopplung
VAR
	pCoupling: POINTER TO HLI_COMMAND_AXIS_COUPLING;
	p_AxisCouplingState: POINTER TO HLI_STATE_AXIS_COUPLING;
	nState: INT;
	bBusy: BOOL;
	fbRTrig: R_TRIG;
	bCouple: BOOL;
	fbFTrig: F_TRIG;
END_VAR

(* allow axis coupling *)
gpAx[5]^.lr_mc_control.axis_coupling.enable_w := TRUE;


pCoupling := ADR(gpAx[5]^.lr_mc_control.axis_coupling.command_w);
p_AxisCouplingState := ADR(gpAx[5]^.lr_mc_control.axis_coupling.state_r);


fbRTrig(clk := bCouple);
fbFTrig(clk := bCouple);


IF (fbRTrig.Q) THEN			(* start coupling *)
	pCoupling^.desc[0].mode  := HLI_AXIS_COUPLING_DIRECT;
	pCoupling^.desc[0].ax_nr := 5;
	bBusy := TRUE;
	nState := 10;
END_IF


IF (fbFTrig.Q) THEN		(* end coupling *)
	pCoupling^.desc[0].mode  := HLI_AXIS_COUPLING_INACTIVE;
	pCoupling^.desc[0].ax_nr := 0;
	bBusy := TRUE;
	nState := 10; 
END_IF




CASE nState OF

0: (*IDLE *)
	bBusy := FALSE;


10: (* Koppeln oder Enkoppeln starten *)
	pCoupling^.semaphor_rw := TRUE;
	nState := nState + 10;

20:	(* Warten auf Koppeln fertig *)
	IF (pCoupling^.semaphor_rw = FALSE) THEN
		nState := 0;
	END_IF


END_CASE

END_PROGRAM

// DUTs/CNC_DataTyps/ITF_ToolAction
INTERFACE ITF_ToolAction

/// Commits the tool data transfer action if it returns true
METHOD Commit : BOOL
VAR_INPUT
	t : ST_CNC_TOOL_DATA_EXT;
END_VAR
END_METHOD

PROPERTY Tool : ST_CNC_TOOL_DATA_EXT
GET
END_GET
END_PROPERTY

END_INTERFACE
